		IF stReciveData.iLength > 0 THEN
			MEMSET(ADR(sReciveMessage),0,SIZEOF(sReciveMessage));
			FUN_TcpBufferDataToString(ADR(sReciveMessage),ADR(stReciveData));
			MEMCPY(ADR(sLastStatusCode),ADR(sReciveMessage),2);
			iLastStatusCode := STRING_TO_INT(sLastStatusCode);
			
			IF iLastStatusCode = 1 THEN 
				eCameraGetConnectionStatus := 1;
				
			ELSIF iLastStatusCode = 0 THEN
				eCameraGetConnectionStatus := 0;
				
			ELSIF iLastStatusCode = -1 THEN
				eCameraGetConnectionStatus := -1;
				
			ELSIF iLastStatusCode = -2 THEN
				eCameraGetConnectionStatus := -2;
				
			ELSIF iLastStatusCode = -6 THEN
				eCameraGetConnectionStatus := -6;
				
			END_IF	
			eCameraMethodState := CAMERA_METHOD_SEND_COMMAND;
			eCameraState := CAMERA_METHOD_DONE;

		END_IF
END_CASE
END_METHOD

METHOD PROTECTED MS_GetExpr
CASE eCameraMethodState OF
	CAMERA_METHOD_SEND_COMMAND:
		MEMSET(ADR(sSendMessage),0,SIZEOF(sSendMessage));
		sSendMessage := FUN_MergeStrings5('Get Expr ',sCellIndexExpr ,CONCAT(TO_STRING(iColumnExpr), TO_STRING(iRowExpr)), '$R$L', '');
		FUN_StringToTcpBufferData(ADR(sSendMessage),ADR(stSendData));
		
		IF fbTcpClient.MR_AppendToSendBuffer(stSendData) THEN
			eCameraMethodState := CAMERA_METHOD_RECEIVE_RESPONSE;
							
		END_IF

	CAMERA_METHOD_RECEIVE_RESPONSE:
		stReciveData := fbTcpClient.NextRecivedMessage;
		
		IF stReciveData.iLength > 0 THEN
			MEMSET(ADR(sReciveMessage),0,SIZEOF(sReciveMessage));
			FUN_TcpBufferDataToString(ADR(sReciveMessage),ADR(stReciveData));
			MEMCPY(ADR(sLastStatusCode),ADR(sReciveMessage),2);
			iLastStatusCode := STRING_TO_INT(sLastStatusCode);
			
			IF iLastStatusCode = 1 THEN 
				eCameraGetExprStatus := 1;
				
			ELSIF iLastStatusCode = 0 THEN
				eCameraGetExprStatus := 0;
				
			ELSIF iLastStatusCode = -1 THEN
				eCameraGetExprStatus := -1;
				
			ELSIF iLastStatusCode = -2 THEN
				eCameraGetExprStatus := -2;
				
			END_IF	
			eCameraMethodState := CAMERA_METHOD_SEND_COMMAND;
			eCameraState := CAMERA_METHOD_DONE;

		END_IF
END_CASE
END_METHOD

METHOD PROTECTED MS_GetFile
CASE eCameraMethodState OF
	CAMERA_METHOD_SEND_COMMAND:
		MEMSET(ADR(sSendMessage),0,SIZEOF(sSendMessage));
		sSendMessage := 'GF$R$L';
		FUN_StringToTcpBufferData(ADR(sSendMessage),ADR(stSendData));
		
		IF fbTcpClient.MR_AppendToSendBuffer(stSendData) THEN
			eCameraMethodState := CAMERA_METHOD_RECEIVE_RESPONSE;
							
		END_IF

	CAMERA_METHOD_RECEIVE_RESPONSE:
		stReciveData := fbTcpClient.NextRecivedMessage;
		
		IF stReciveData.iLength > 0 THEN
			MEMSET(ADR(sReciveMessage),0,SIZEOF(sReciveMessage));
			FUN_TcpBufferDataToString(ADR(sReciveMessage),ADR(stReciveData));
			MEMCPY(ADR(sLastStatusCode),ADR(sReciveMessage),2);
			iLastStatusCode := STRING_TO_INT(sLastStatusCode);
			
			IF iLastStatusCode = 1 THEN 
				eCameraGetFileStatus := 1;
				
			ELSIF iLastStatusCode = 0 THEN
				eCameraGetFileStatus := 0;
				
			ELSIF iLastStatusCode = -2 THEN
				eCameraGetFileStatus := -2;
				
			END_IF	
			eCameraMethodState := CAMERA_METHOD_SEND_COMMAND;
			eCameraState := CAMERA_METHOD_DONE;

		END_IF
END_CASE
END_METHOD

METHOD PROTECTED MS_GetFileList
CASE eCameraMethodState OF
	CAMERA_METHOD_SEND_COMMAND:
		MEMSET(ADR(sSendMessage),0,SIZEOF(sSendMessage));
		sSendMessage := 'Get Filelist$R$L';
		FUN_StringToTcpBufferData(ADR(sSendMessage),ADR(stSendData));
		
		IF fbTcpClient.MR_AppendToSendBuffer(stSendData) THEN
			eCameraMethodState := CAMERA_METHOD_RECEIVE_RESPONSE;
							
		END_IF

	CAMERA_METHOD_RECEIVE_RESPONSE:
		stReciveData := fbTcpClient.NextRecivedMessage;
		
		IF stReciveData.iLength > 0 THEN
			MEMSET(ADR(sReciveMessage),0,SIZEOF(sReciveMessage));
			FUN_TcpBufferDataToString(ADR(sReciveMessage),ADR(stReciveData));
			MEMCPY(ADR(sLastStatusCode),ADR(sReciveMessage),2);
			iLastStatusCode := STRING_TO_INT(sLastStatusCode);
			
			IF iLastStatusCode = 1 THEN 
				eCameraGetFileListStatus := 1;
				
			ELSIF iLastStatusCode = 0 THEN
				eCameraGetFileListStatus := 0;
				
			ELSIF iLastStatusCode = -1 THEN
				eCameraGetFileListStatus := -1;
				
			ELSIF iLastStatusCode = -2 THEN
				eCameraGetFileListStatus := -2;
				
			END_IF	
			eCameraMethodState := CAMERA_METHOD_SEND_COMMAND;
			eCameraState := CAMERA_METHOD_DONE;

		END_IF
END_CASE
END_METHOD

METHOD PROTECTED MS_GetJob
CASE eCameraMethodState OF
	CAMERA_METHOD_SEND_COMMAND:
		MEMSET(ADR(sSendMessage),0,SIZEOF(sSendMessage));
		sSendMessage := 'GJ$R$L';
		FUN_StringToTcpBufferData(ADR(sSendMessage),ADR(stSendData));
		
		IF fbTcpClient.MR_AppendToSendBuffer(stSendData) THEN
			eCameraMethodState := CAMERA_METHOD_RECEIVE_RESPONSE;
							
		END_IF

	CAMERA_METHOD_RECEIVE_RESPONSE:
		stReciveData := fbTcpClient.NextRecivedMessage;
		
		IF stReciveData.iLength > 0 THEN
			MEMSET(ADR(sReciveMessage),0,SIZEOF(sReciveMessage));
			FUN_TcpBufferDataToString(ADR(sReciveMessage),ADR(stReciveData));
			MEMCPY(ADR(sLastStatusCode),ADR(sReciveMessage),2);
			iLastStatusCode := STRING_TO_INT(sLastStatusCode);
			
			IF iLastStatusCode = 1 THEN 
				eCameraGetJobStatus := 1;
				
			ELSIF iLastStatusCode = 0 THEN
				eCameraGetJobStatus := 0;
				
			ELSIF iLastStatusCode = -2 THEN
				eCameraGetJobStatus := -2;
				
			END_IF	
			eCameraMethodState := CAMERA_METHOD_SEND_COMMAND;
			eCameraState := CAMERA_METHOD_DONE;

		END_IF
END_CASE
END_METHOD

METHOD PROTECTED MS_GetOnline
CASE eCameraMethodState OF
	CAMERA_METHOD_SEND_COMMAND:
		MEMSET(ADR(sSendMessage),0,SIZEOF(sSendMessage));
		sSendMessage := 'GO$R$L';
		FUN_StringToTcpBufferData(ADR(sSendMessage),ADR(stSendData));
		
		IF fbTcpClient.MR_AppendToSendBuffer(stSendData) THEN
			eCameraMethodState := CAMERA_METHOD_RECEIVE_RESPONSE;
							
		END_IF

	CAMERA_METHOD_RECEIVE_RESPONSE:
		stReciveData := fbTcpClient.NextRecivedMessage;
		
		IF stReciveData.iLength > 0 THEN
			MEMSET(ADR(sReciveMessage),0,SIZEOF(sReciveMessage));
			FUN_TcpBufferDataToString(ADR(sReciveMessage),ADR(stReciveData));
			MEMCPY(ADR(sLastStatusCode),ADR(sReciveMessage),2);
			iLastStatusCode := STRING_TO_INT(sLastStatusCode);
			
			IF iLastStatusCode = 0 THEN 
				eCameraGetOnlineStatus := 0;
				
			ELSIF iLastStatusCode = 1 THEN
				eCameraGetOnlineStatus := 1;
				
			END_IF	
			eCameraMethodState := CAMERA_METHOD_SEND_COMMAND;
			eCameraState := CAMERA_METHOD_DONE;

		END_IF
END_CASE
END_METHOD

METHOD PROTECTED MS_GetPosition
CASE eCameraGetPositionState OF
	CAMERA_GET_POSITION_SEND_COMMAND_X:
		MEMSET(ADR(sSendMessage),0,SIZEOF(sSendMessage));
		sSendMessage := FUN_MergeStrings3('GV', sPositionXVariable,'$R$L');
		FUN_StringToTcpBufferData(ADR(sSendMessage),ADR(stSendData));
		
		IF fbTcpClient.MR_AppendToSendBuffer(stSendData) THEN
			eCameraGetPositionState := CAMERA_GET_POSITION_RECEIVE_RESPONSE_X;
							
		END_IF

	CAMERA_GET_POSITION_RECEIVE_RESPONSE_X:
		stReciveData := fbTcpClient.NextRecivedMessage;
		
		IF stReciveData.iLength > 0 THEN
			MEMSET(ADR(sReciveMessage),0,SIZEOF(sReciveMessage));
			FUN_TcpBufferDataToString(ADR(sReciveMessage),ADR(stReciveData));
			MEMCPY(ADR(sLastStatusCode),ADR(sReciveMessage),2);
			iLastStatusCode := STRING_TO_INT(sLastStatusCode);
			
			IF iLastStatusCode = 1 THEN 
				eCameraGetPositionStatus := 1;
				sPositionString := TO_STRING(sReciveMessage);
				sPositionStringDel := DELETE(sPositionString,3,1);
				lrPositionX := STRING_TO_LREAL(sPositionStringDel);
				
			ELSIF iLastStatusCode = 0 THEN
				eCameraGetPositionStatus := 0;
				
			ELSIF iLastStatusCode = -1 THEN
				eCameraGetPositionStatus := -1;
				
			ELSIF iLastStatusCode = -2 THEN
				eCameraGetPositionStatus := -2;
				
			END_IF	
			eCameraGetPositionState := CAMERA_GET_POSITION_SEND_COMMAND_Y;

		END_IF
	
	CAMERA_GET_POSITION_SEND_COMMAND_Y:
		MEMSET(ADR(sSendMessage),0,SIZEOF(sSendMessage));
		sSendMessage := FUN_MergeStrings3('GV', sPositionYVariable,'$R$L');
		FUN_StringToTcpBufferData(ADR(sSendMessage),ADR(stSendData));
		
		IF fbTcpClient.MR_AppendToSendBuffer(stSendData) THEN
			eCameraGetPositionState := CAMERA_GET_POSITION_RECEIVE_RESPONSE_Y;
							
		END_IF

	CAMERA_GET_POSITION_RECEIVE_RESPONSE_Y:
		stReciveData := fbTcpClient.NextRecivedMessage;
		
		IF stReciveData.iLength > 0 THEN
			MEMSET(ADR(sReciveMessage),0,SIZEOF(sReciveMessage));
			FUN_TcpBufferDataToString(ADR(sReciveMessage),ADR(stReciveData));
			MEMCPY(ADR(sLastStatusCode),ADR(sReciveMessage),2);
			iLastStatusCode := STRING_TO_INT(sLastStatusCode);
			
			IF iLastStatusCode = 1 THEN 
				eCameraGetPositionStatus := 1;
				sPositionString := TO_STRING(sReciveMessage);
				sPositionStringDel := DELETE(sPositionString,3,1);
				lrPositionY := STRING_TO_LREAL(sPositionStringDel);
				
			ELSIF iLastStatusCode = 0 THEN
				eCameraGetPositionStatus := 0;
				
			ELSIF iLastStatusCode = -1 THEN
				eCameraGetPositionStatus := -1;
				
			ELSIF iLastStatusCode = -2 THEN
				eCameraGetPositionStatus := -2;
				
			END_IF	
			eCameraGetPositionState := CAMERA_GET_POSITION_SEND_COMMAND_ROTATION;
			
		END_IF
		
		
	CAMERA_GET_POSITION_SEND_COMMAND_ROTATION:
		MEMSET(ADR(sSendMessage),0,SIZEOF(sSendMessage));
		sSendMessage := FUN_MergeStrings3('GV', sRotationVariable,'$R$L');
		FUN_StringToTcpBufferData(ADR(sSendMessage),ADR(stSendData));
		
		IF fbTcpClient.MR_AppendToSendBuffer(stSendData) THEN
			eCameraGetPositionState := CAMERA_GET_POSITION_RECEIVE_RESPONSE_ROTATION;
							
		END_IF

	CAMERA_GET_POSITION_RECEIVE_RESPONSE_ROTATION:
		stReciveData := fbTcpClient.NextRecivedMessage;
		
		IF stReciveData.iLength > 0 THEN
			MEMSET(ADR(sReciveMessage),0,SIZEOF(sReciveMessage));
			FUN_TcpBufferDataToString(ADR(sReciveMessage),ADR(stReciveData));
			MEMCPY(ADR(sLastStatusCode),ADR(sReciveMessage),2);
			iLastStatusCode := STRING_TO_INT(sLastStatusCode);
			
			IF iLastStatusCode = 1 THEN 
				eCameraGetPositionStatus := 1;
				sPositionString := TO_STRING(sReciveMessage);
				sPositionStringDel := DELETE(sPositionString,3,1);
				lrRotation := STRING_TO_LREAL(sPositionStringDel);
				
			ELSIF iLastStatusCode = 0 THEN
				eCameraGetPositionStatus := 0;
				
			ELSIF iLastStatusCode = -1 THEN
				eCameraGetPositionStatus := -1;
				
			ELSIF iLastStatusCode = -2 THEN
				eCameraGetPositionStatus := -2;
				
			END_IF	
			eCameraGetPositionState := CAMERA_GET_POSITION_GETTING_DONE;

		END_IF
		
	CAMERA_GET_POSITION_GETTING_DONE:
		IF lrPositionX = 0.0 AND lrPositionY = 0.0 THEN
			eCameraGetPositionStatus := -3;
			
		END_IF
		eCameraGetPositionState := CAMERA_GET_POSITION_SEND_COMMAND_X;
		eCameraState := CAMERA_METHOD_DONE;
		
END_CASE
END_METHOD

METHOD PROTECTED MS_GetValueEasyBuilder
CASE eCameraMethodState OF
	CAMERA_METHOD_SEND_COMMAND:
		MEMSET(ADR(sSendMessage),0,SIZEOF(sSendMessage));
		sSendMessage := FUN_MergeStrings3('GV', sEasyBuilderValueName,'$R$L');
		FUN_StringToTcpBufferData(ADR(sSendMessage),ADR(stSendData));
		
		IF fbTcpClient.MR_AppendToSendBuffer(stSendData) THEN
			eCameraMethodState := CAMERA_METHOD_RECEIVE_RESPONSE;
							
		END_IF

	CAMERA_METHOD_RECEIVE_RESPONSE:
		stReciveData := fbTcpClient.NextRecivedMessage;
		
		IF stReciveData.iLength > 0 THEN
			MEMSET(ADR(sReciveMessage),0,SIZEOF(sReciveMessage));
			FUN_TcpBufferDataToString(ADR(sReciveMessage),ADR(stReciveData));
			MEMCPY(ADR(sLastStatusCode),ADR(sReciveMessage),2);
			iLastStatusCode := STRING_TO_INT(sLastStatusCode);
			
			IF iLastStatusCode = 1 THEN 
				eCameraGetValueEasyBuilderStatus := 1;
				
			ELSIF iLastStatusCode = 0 THEN
				eCameraGetValueEasyBuilderStatus := 0;
				
			ELSIF iLastStatusCode = -1 THEN
				eCameraGetValueEasyBuilderStatus := -1;
				
			ELSIF iLastStatusCode = -2 THEN
				eCameraGetValueEasyBuilderStatus := -2;
				
			END_IF	
			eCameraMethodState := CAMERA_METHOD_SEND_COMMAND;
			eCameraState := CAMERA_METHOD_DONE;

		END_IF
END_CASE
END_METHOD

METHOD PROTECTED MS_GetValues
CASE eCameraGetValuesState OF
	CAMERA_GET_VALUES_SEND_COMMAND_VALUE_1:
		MEMSET(ADR(sSendMessage),0,SIZEOF(sSendMessage));
		sSendMessage := FUN_MergeStrings3('GV', sVariable1,'$R$L');
		FUN_StringToTcpBufferData(ADR(sSendMessage),ADR(stSendData));
		
		IF fbTcpClient.MR_AppendToSendBuffer(stSendData) THEN
			eCameraGetValuesState := CAMERA_GET_VALUES_RECEIVE_RESPONSE_VALUE_1;
							
		END_IF

	CAMERA_GET_VALUES_RECEIVE_RESPONSE_VALUE_1:
		stReciveData := fbTcpClient.NextRecivedMessage;
		
		IF stReciveData.iLength > 0 THEN
			MEMSET(ADR(sReciveMessage),0,SIZEOF(sReciveMessage));
			FUN_TcpBufferDataToString(ADR(sReciveMessage),ADR(stReciveData));
			MEMCPY(ADR(sLastStatusCode),ADR(sReciveMessage),2);
			iLastStatusCode := STRING_TO_INT(sLastStatusCode);
			
			IF iLastStatusCode = 1 THEN 
				eCameraGetValuesStatus := 1;
				sPositionString := TO_STRING(sReciveMessage);
				sPositionStringDel := DELETE(sPositionString,3,1);
				lrValue1 := STRING_TO_LREAL(sPositionStringDel);
				
			ELSIF iLastStatusCode = 0 THEN
				eCameraGetValuesStatus := 0;
				
			ELSIF iLastStatusCode = -1 THEN
				eCameraGetValuesStatus := -1;
				
			ELSIF iLastStatusCode = -2 THEN
				eCameraGetValuesStatus := -2;
				
			END_IF	
			eCameraGetValuesState := CAMERA_GET_VALUES_SEND_COMMAND_VALUE_2;

		END_IF
	
	CAMERA_GET_VALUES_SEND_COMMAND_VALUE_2:
		MEMSET(ADR(sSendMessage),0,SIZEOF(sSendMessage));
		sSendMessage := FUN_MergeStrings3('GV', sVariable2,'$R$L');
		FUN_StringToTcpBufferData(ADR(sSendMessage),ADR(stSendData));
		
		IF fbTcpClient.MR_AppendToSendBuffer(stSendData) THEN
			eCameraGetValuesState := CAMERA_GET_VALUES_RECEIVE_RESPONSE_VALUE_2;
							
		END_IF

	CAMERA_GET_VALUES_RECEIVE_RESPONSE_VALUE_2:
		stReciveData := fbTcpClient.NextRecivedMessage;
		
		IF stReciveData.iLength > 0 THEN
			MEMSET(ADR(sReciveMessage),0,SIZEOF(sReciveMessage));
			FUN_TcpBufferDataToString(ADR(sReciveMessage),ADR(stReciveData));
			MEMCPY(ADR(sLastStatusCode),ADR(sReciveMessage),2);
			iLastStatusCode := STRING_TO_INT(sLastStatusCode);
			
			IF iLastStatusCode = 1 THEN 
				eCameraGetValuesStatus := 1;
				sPositionString := TO_STRING(sReciveMessage);
				sPositionStringDel := DELETE(sPositionString,3,1);
				lrValue2 := STRING_TO_LREAL(sPositionStringDel);
				
			ELSIF iLastStatusCode = 0 THEN
				eCameraGetValuesStatus := 0;
				
			ELSIF iLastStatusCode = -1 THEN
				eCameraGetValuesStatus := -1;
				
			ELSIF iLastStatusCode = -2 THEN
				eCameraGetValuesStatus := -2;
				
			END_IF	
			eCameraGetValuesState := CAMERA_GET_VALUES_SEND_COMMAND_VALUE_3;
			
		END_IF
		
		
	CAMERA_GET_VALUES_SEND_COMMAND_VALUE_3:
		MEMSET(ADR(sSendMessage),0,SIZEOF(sSendMessage));
		sSendMessage := FUN_MergeStrings3('GV', sVariable3,'$R$L');
		FUN_StringToTcpBufferData(ADR(sSendMessage),ADR(stSendData));
		
		IF fbTcpClient.MR_AppendToSendBuffer(stSendData) THEN
			eCameraGetValuesState := CAMERA_GET_VALUES_RECEIVE_RESPONSE_VALUE_3;

		END_IF

	CAMERA_GET_VALUES_RECEIVE_RESPONSE_VALUE_3:
		stReciveData := fbTcpClient.NextRecivedMessage;
		
		IF stReciveData.iLength > 0 THEN
			MEMSET(ADR(sReciveMessage),0,SIZEOF(sReciveMessage));
			FUN_TcpBufferDataToString(ADR(sReciveMessage),ADR(stReciveData));
			MEMCPY(ADR(sLastStatusCode),ADR(sReciveMessage),2);
			iLastStatusCode := STRING_TO_INT(sLastStatusCode);
			
			IF iLastStatusCode = 1 THEN 
				eCameraGetValuesStatus := 1;
				sPositionString := TO_STRING(sReciveMessage);
				sPositionStringDel := DELETE(sPositionString,3,1);
				lrValue3 := STRING_TO_LREAL(sPositionStringDel);
				
			ELSIF iLastStatusCode = 0 THEN
				eCameraGetValuesStatus := 0;
				
			ELSIF iLastStatusCode = -1 THEN
				eCameraGetValuesStatus := -1;
				
			ELSIF iLastStatusCode = -2 THEN
				eCameraGetValuesStatus := -2;
				
			END_IF	
			eCameraGetValuesState := CAMERA_GET_VALUES_SEND_COMMAND_VALUE_4;

		END_IF


	CAMERA_GET_VALUES_SEND_COMMAND_VALUE_4:
		MEMSET(ADR(sSendMessage),0,SIZEOF(sSendMessage));
		sSendMessage := FUN_MergeStrings3('GV', sVariable4,'$R$L');
		FUN_StringToTcpBufferData(ADR(sSendMessage),ADR(stSendData));
		
		IF fbTcpClient.MR_AppendToSendBuffer(stSendData) THEN
			eCameraGetValuesState := CAMERA_GET_VALUES_RECEIVE_RESPONSE_VALUE_4;
							
		END_IF

	CAMERA_GET_VALUES_RECEIVE_RESPONSE_VALUE_4:
		stReciveData := fbTcpClient.NextRecivedMessage;
		
		IF stReciveData.iLength > 0 THEN
			MEMSET(ADR(sReciveMessage),0,SIZEOF(sReciveMessage));
			FUN_TcpBufferDataToString(ADR(sReciveMessage),ADR(stReciveData));
			MEMCPY(ADR(sLastStatusCode),ADR(sReciveMessage),2);
			iLastStatusCode := STRING_TO_INT(sLastStatusCode);
			
			IF iLastStatusCode = 1 THEN 
				eCameraGetValuesStatus := 1;
				sPositionString := TO_STRING(sReciveMessage);
				sPositionStringDel := DELETE(sPositionString,3,1);
				lrValue4 := STRING_TO_LREAL(sPositionStringDel);
				
			ELSIF iLastStatusCode = 0 THEN
				eCameraGetValuesStatus := 0;
				
			ELSIF iLastStatusCode = -1 THEN
				eCameraGetValuesStatus := -1;
				
			ELSIF iLastStatusCode = -2 THEN
				eCameraGetValuesStatus := -2;
				
			END_IF	
			eCameraGetValuesState := CAMERA_GET_VALUES_GETTING_DONE;

		END_IF
		
	CAMERA_GET_VALUES_GETTING_DONE:
		
		IF lrValue1 = 0.0 OR lrValue2 = 0.0 OR lrValue3 = 0.0 OR lrValue4 = 0.0 THEN
			eCameraGetValuesStatus := -3;
			
		END_IF
		eCameraGetValuesState := CAMERA_GET_VALUES_SEND_COMMAND_VALUE_1;
		eCameraState := CAMERA_METHOD_DONE;
		
END_CASE
END_METHOD

METHOD PROTECTED MS_GetValueSpreadsheet
CASE eCameraMethodState OF
	CAMERA_METHOD_SEND_COMMAND:
		MEMSET(ADR(sSendMessage),0,SIZEOF(sSendMessage));
		sSendMessage := FUN_MergeStrings5('GV', TO_STRING(iColumnValueSpreadsheet), TO_STRING(iRowValueSpreadsheet), '$R$L', '');
		FUN_StringToTcpBufferData(ADR(sSendMessage),ADR(stSendData));
		
		IF fbTcpClient.MR_AppendToSendBuffer(stSendData) THEN
			eCameraMethodState := CAMERA_METHOD_RECEIVE_RESPONSE;
							
		END_IF

	CAMERA_METHOD_RECEIVE_RESPONSE:
		stReciveData := fbTcpClient.NextRecivedMessage;
		
		IF stReciveData.iLength > 0 THEN
			MEMSET(ADR(sReciveMessage),0,SIZEOF(sReciveMessage));
			FUN_TcpBufferDataToString(ADR(sReciveMessage),ADR(stReciveData));
			MEMCPY(ADR(sLastStatusCode),ADR(sReciveMessage),2);
			iLastStatusCode := STRING_TO_INT(sLastStatusCode);
			
			IF iLastStatusCode = 1 THEN 
				eCameraGetValueSpreadsheetStatus := 1;
				
			ELSIF iLastStatusCode = 0 THEN
				eCameraGetValueSpreadsheetStatus := 0;
				
			ELSIF iLastStatusCode = -1 THEN
				eCameraGetValueSpreadsheetStatus := -1;
				
			ELSIF iLastStatusCode = -2 THEN
				eCameraGetValueSpreadsheetStatus := -2;
				
			END_IF	
			eCameraMethodState := CAMERA_METHOD_SEND_COMMAND;
			eCameraState := CAMERA_METHOD_DONE;

		END_IF
END_CASE
END_METHOD

METHOD PROTECTED MS_Idle
;
END_METHOD

METHOD PROTECTED MS_ImageTrigger
CASE eCameraMethodState OF
	CAMERA_METHOD_SEND_COMMAND:
		MEMSET(ADR(sSendMessage),0,SIZEOF(sSendMessage));
		sSendMessage := 'SW8$R$L';
		FUN_StringToTcpBufferData(ADR(sSendMessage),ADR(stSendData));
		
		IF fbTcpClient.MR_AppendToSendBuffer(stSendData) THEN
			eCameraMethodState := CAMERA_METHOD_RECEIVE_RESPONSE;
							
		END_IF

	CAMERA_METHOD_RECEIVE_RESPONSE:
		stReciveData := fbTcpClient.NextRecivedMessage;
		
		IF stReciveData.iLength > 0 THEN
			MEMSET(ADR(sReciveMessage),0,SIZEOF(sReciveMessage));
			FUN_TcpBufferDataToString(ADR(sReciveMessage),ADR(stReciveData));
			MEMCPY(ADR(sLastStatusCode),ADR(sReciveMessage),2);
			iLastStatusCode := STRING_TO_INT(sLastStatusCode);
			
			IF iLastStatusCode = 1 THEN 
				eCameraImageTriggerStatus := 1;
				
			ELSIF iLastStatusCode = 0 THEN
				eCameraImageTriggerStatus := 0;
				
			ELSIF iLastStatusCode = -1 THEN
				eCameraImageTriggerStatus := -1;
				
			ELSIF iLastStatusCode = -2 THEN
				eCameraImageTriggerStatus := -2;
				
			ELSIF iLastStatusCode = -6 THEN
				eCameraImageTriggerStatus := -6;
				
			END_IF	
			eCameraMethodState := CAMERA_METHOD_SEND_COMMAND;			
			eCameraState := CAMERA_METHOD_DONE;

		END_IF
END_CASE
END_METHOD

METHOD PROTECTED MS_Initializing //C:\TwinCAT\log\filelog.txt
VAR_INST
//	tClearBuffers		:	TON;
END_VAR
CASE eCameraInitState OF
	CAMERA_INIT_CONNECTION:
		fbTcpClient.MR_Init();
		
		IF fbTcpClient.Active THEN
			eCameraInitState := CAMERA_INIT_CLEAR_BUFFER;	
			
		ELSIF fbTcpClient.Error THEN
			bError := TRUE;
			iErrorID := fbTcpClient.ErrorID;
			
		END_IF
		
	CAMERA_INIT_CLEAR_BUFFER:
		fbTcpClient.MR_ClearAllBuffers();
		eCameraInitState := CAMERA_INIT_WAIT_FOR_USERNAME;
		
		IF fbTcpClient.Error THEN
			bError := TRUE;
			iErrorID := fbTcpClient.ErrorID;
			
		END_IF
		
	CAMERA_INIT_WAIT_FOR_USERNAME: 
		stReciveData := fbTcpClient.NextRecivedMessage;
		
		IF stReciveData.iLength > 0 THEN
			MEMSET(ADR(sReciveMessage),0,SIZEOF(sReciveMessage));
			FUN_TcpBufferDataToString(ADR(sReciveMessage),ADR(stReciveData));		
	
			IF RIGHT(sReciveMessage, 6) = 'User: ' THEN	
				eCameraInitState := CAMERA_INIT_WRITE_USER;
			
			END_IF
		ELSIF fbTcpClient.Error THEN
			bError := TRUE;
			iErrorID := fbTcpClient.ErrorID;
			
		END_IF
			
	CAMERA_INIT_WRITE_USER:
		MEMSET(ADR(sSendMessage),0,SIZEOF(sSendMessage));
		sSendMessage := 'admin$R$L';
		FUN_StringToTcpBufferData(ADR(sSendMessage),ADR(stSendData));
		stSendData.iLength := INT_TO_UDINT(LEN(sSendMessage));
		
		IF fbTcpClient.MR_AppendToSendBuffer(stSendData) THEN
			eCameraInitState := CAMERA_INIT_WAIT_FOR_PASSWORD;
		
		ELSIF fbTcpClient.Error THEN
			bError := TRUE;
			iErrorID := fbTcpClient.ErrorID;
			
		END_IF
		
	CAMERA_INIT_WAIT_FOR_PASSWORD:
		stReciveData := fbTcpClient.NextRecivedMessage;
		
		IF stReciveData.iLength > 0 THEN
			MEMSET(ADR(sReciveMessage),0,SIZEOF(sReciveMessage));
			FUN_TcpBufferDataToString(ADR(sReciveMessage),ADR(stReciveData));
			
			IF sReciveMessage = 'Password: ' THEN		
				eCameraInitState := CAMERA_INIT_WRITE_PASSWORD;
			
			END_IF
		ELSIF fbTcpClient.Error THEN
			bError := TRUE;
			iErrorID := fbTcpClient.ErrorID;
			
		END_IF

	CAMERA_INIT_WRITE_PASSWORD:
		MEMSET(ADR(sSendMessage),0,SIZEOF(sSendMessage));
		sSendMessage := '$R$L';
		FUN_StringToTcpBufferData(ADR(sSendMessage),ADR(stSendData));
		stSendData.iLength := INT_TO_UDINT(LEN(sSendMessage));
		
		IF fbTcpClient.MR_AppendToSendBuffer(stSendData) THEN
			eCameraInitState := CAMERA_INIT_WAIT_FOR_CONFIRMATION;

		ELSIF fbTcpClient.Error THEN
			bError := TRUE;
			iErrorID := fbTcpClient.ErrorID;
			
		END_IF
		
	CAMERA_INIT_WAIT_FOR_CONFIRMATION:
		stReciveData := fbTcpClient.NextRecivedMessage;
		
		IF stReciveData.iLength > 0 THEN
			MEMSET(ADR(sReciveMessage),0,SIZEOF(sReciveMessage));
			FUN_TcpBufferDataToString(ADR(sReciveMessage),ADR(stReciveData));
	
			IF sReciveMessage = 'User Logged In$R$L' THEN		
				eCameraInitState := CAMERA_INIT_DONE;
			
			END_IF
		ELSIF fbTcpClient.Error THEN
			bError := TRUE;
			iErrorID := fbTcpClient.ErrorID;
			
		END_IF
		
	CAMERA_INIT_DONE:
		eCameraInitState := CAMERA_INIT_CONNECTION;
		eCameraState := CAMERA_READY;
			
END_CASE
END_METHOD

METHOD PROTECTED MS_LoadFile
CASE eCameraMethodState OF
	CAMERA_METHOD_SEND_COMMAND:
		MEMSET(ADR(sSendMessage),0,SIZEOF(sSendMessage));
		sSendMessage := FUN_MergeStrings3('LF', sLoadFileName,'$R$L');
		FUN_StringToTcpBufferData(ADR(sSendMessage),ADR(stSendData));
		
		IF fbTcpClient.MR_AppendToSendBuffer(stSendData) THEN
			eCameraMethodState := CAMERA_METHOD_RECEIVE_RESPONSE;
							
		END_IF

	CAMERA_METHOD_RECEIVE_RESPONSE:
		stReciveData := fbTcpClient.NextRecivedMessage;
		
		IF stReciveData.iLength > 0 THEN
			MEMSET(ADR(sReciveMessage),0,SIZEOF(sReciveMessage));
			FUN_TcpBufferDataToString(ADR(sReciveMessage),ADR(stReciveData));
			MEMCPY(ADR(sLastStatusCode),ADR(sReciveMessage),2);
			iLastStatusCode := STRING_TO_INT(sLastStatusCode);
			
			IF iLastStatusCode = 1 THEN 
				eCameraLoadFileStatus := 1;
				
			ELSIF iLastStatusCode = 0 THEN
				eCameraLoadFileStatus := 0;
				
			ELSIF iLastStatusCode = -1 THEN
				eCameraLoadFileStatus := -1;
				
			ELSIF iLastStatusCode = -2 THEN
				eCameraLoadFileStatus := -2;
				
			ELSIF iLastStatusCode = -4 THEN
				eCameraLoadFileStatus := -4;
				
			ELSIF iLastStatusCode = -6 THEN
				eCameraLoadFileStatus := -6;
				
			END_IF	
			eCameraMethodState := CAMERA_METHOD_SEND_COMMAND;
			eCameraState := CAMERA_METHOD_DONE;

		END_IF
END_CASE
END_METHOD

METHOD PROTECTED MS_MethodDone
VAR_INPUT
END_VAR
IF NOT bBusy THEN
	eCameraState := CAMERA_IDLE;
	
END_IF
END_METHOD

METHOD PROTECTED MS_PutLive
CASE eCameraMethodState OF
	CAMERA_METHOD_SEND_COMMAND:
		MEMSET(ADR(sSendMessage),0,SIZEOF(sSendMessage));
		sSendMessage := FUN_MergeStrings3('Put live ', TO_STRING(bEnableLiveAcquisition), '$R$L');
		FUN_StringToTcpBufferData(ADR(sSendMessage),ADR(stSendData));
		
		IF fbTcpClient.MR_AppendToSendBuffer(stSendData) THEN
			eCameraMethodState := CAMERA_METHOD_RECEIVE_RESPONSE;
							
		END_IF

	CAMERA_METHOD_RECEIVE_RESPONSE:
		stReciveData := fbTcpClient.NextRecivedMessage;
		
		IF stReciveData.iLength > 0 THEN
			MEMSET(ADR(sReciveMessage),0,SIZEOF(sReciveMessage));
			FUN_TcpBufferDataToString(ADR(sReciveMessage),ADR(stReciveData));
			MEMCPY(ADR(sLastStatusCode),ADR(sReciveMessage),2);
			iLastStatusCode := STRING_TO_INT(sLastStatusCode);
			
			IF iLastStatusCode = 1 THEN 
				eCameraPutLiveStatus := 1;
				
			ELSIF iLastStatusCode = 0 THEN
				eCameraPutLiveStatus := 0;
				
			ELSIF iLastStatusCode = -1 THEN
				eCameraPutLiveStatus := -1;
				
			ELSIF iLastStatusCode = -2 THEN
				eCameraPutLiveStatus := -2;
				
			ELSIF iLastStatusCode = -6 THEN
				eCameraPutLiveStatus := -6;
				
			END_IF	
			eCameraMethodState := CAMERA_METHOD_SEND_COMMAND;
			eCameraState := CAMERA_METHOD_DONE;

		END_IF
END_CASE
END_METHOD

METHOD PROTECTED MS_PutPortnum
CASE eCameraMethodState OF
	CAMERA_METHOD_SEND_COMMAND:
		MEMSET(ADR(sSendMessage),0,SIZEOF(sSendMessage));
		sSendMessage := FUN_MergeStrings3('Put Portnum ', TO_STRING(iPortNumber), '$R$L');
		FUN_StringToTcpBufferData(ADR(sSendMessage),ADR(stSendData));
		
		IF fbTcpClient.MR_AppendToSendBuffer(stSendData) THEN
			eCameraMethodState := CAMERA_METHOD_RECEIVE_RESPONSE;
							
		END_IF

	CAMERA_METHOD_RECEIVE_RESPONSE:
		stReciveData := fbTcpClient.NextRecivedMessage;
		
		IF stReciveData.iLength > 0 THEN
			MEMSET(ADR(sReciveMessage),0,SIZEOF(sReciveMessage));
			FUN_TcpBufferDataToString(ADR(sReciveMessage),ADR(stReciveData));
			MEMCPY(ADR(sLastStatusCode),ADR(sReciveMessage),2);
			iLastStatusCode := STRING_TO_INT(sLastStatusCode);
			
			IF iLastStatusCode = 1 THEN 
				eCameraPutPortnumStatus := 1;
				
			ELSIF iLastStatusCode = 0 THEN
				eCameraPutPortnumStatus := 0;
				
			ELSIF iLastStatusCode = -1 THEN
				eCameraPutPortnumStatus := -1;
				
			ELSIF iLastStatusCode = -2 THEN
				eCameraPutPortnumStatus := -2;
				
			ELSIF iLastStatusCode = -6 THEN
				eCameraPutPortnumStatus := -6;
				
			END_IF	
			eCameraMethodState := CAMERA_METHOD_SEND_COMMAND;
			eCameraState := CAMERA_METHOD_DONE;

		END_IF
END_CASE
END_METHOD

METHOD PROTECTED MS_PutTimeout
CASE eCameraMethodState OF
	CAMERA_METHOD_SEND_COMMAND:
		MEMSET(ADR(sSendMessage),0,SIZEOF(sSendMessage));
		sSendMessage := FUN_MergeStrings3('Put Timeout ', TO_STRING(iTimeout), '$R$L');
		FUN_StringToTcpBufferData(ADR(sSendMessage),ADR(stSendData));
		
		IF fbTcpClient.MR_AppendToSendBuffer(stSendData) THEN
			eCameraMethodState := CAMERA_METHOD_RECEIVE_RESPONSE;
							
		END_IF

	CAMERA_METHOD_RECEIVE_RESPONSE:
		stReciveData := fbTcpClient.NextRecivedMessage;
		
		IF stReciveData.iLength > 0 THEN
			MEMSET(ADR(sReciveMessage),0,SIZEOF(sReciveMessage));
			FUN_TcpBufferDataToString(ADR(sReciveMessage),ADR(stReciveData));
			MEMCPY(ADR(sLastStatusCode),ADR(sReciveMessage),2);
			iLastStatusCode := STRING_TO_INT(sLastStatusCode);
			
			IF iLastStatusCode = 1 THEN 
				eCameraPutTimeoutStatus := 1;
				
			ELSIF iLastStatusCode = 0 THEN
				eCameraPutTimeoutStatus := 0;
				
			ELSIF iLastStatusCode = -1 THEN
				eCameraPutTimeoutStatus := -1;
				
			ELSIF iLastStatusCode = -6 THEN
				eCameraPutTimeoutStatus := -6;
				
			END_IF	
			eCameraMethodState := CAMERA_METHOD_SEND_COMMAND;
			eCameraState := CAMERA_METHOD_DONE;
			
		END_IF
END_CASE
END_METHOD

METHOD PROTECTED MS_PutUpdate
CASE eCameraMethodState OF
	CAMERA_METHOD_SEND_COMMAND:
		MEMSET(ADR(sSendMessage),0,SIZEOF(sSendMessage));
		sSendMessage := FUN_MergeStrings3('Put Update ', TO_STRING(iUpdateNumber), '$R$L');
		FUN_StringToTcpBufferData(ADR(sSendMessage),ADR(stSendData));
		
		IF fbTcpClient.MR_AppendToSendBuffer(stSendData) THEN
			eCameraMethodState := CAMERA_METHOD_RECEIVE_RESPONSE;
							
		END_IF

	CAMERA_METHOD_RECEIVE_RESPONSE:
		stReciveData := fbTcpClient.NextRecivedMessage;
		
		IF stReciveData.iLength > 0 THEN
			MEMSET(ADR(sReciveMessage),0,SIZEOF(sReciveMessage));
			FUN_TcpBufferDataToString(ADR(sReciveMessage),ADR(stReciveData));
			MEMCPY(ADR(sLastStatusCode),ADR(sReciveMessage),2);
			iLastStatusCode := STRING_TO_INT(sLastStatusCode);
			
			IF iLastStatusCode = 1 THEN 
				eCameraPutUpdateStatus := 1;
				
			ELSIF iLastStatusCode = 0 THEN
				eCameraPutUpdateStatus := 0;
				
			ELSIF iLastStatusCode = -1 THEN
				eCameraPutUpdateStatus := -1;
				
			ELSIF iLastStatusCode = -2 THEN
				eCameraPutUpdateStatus := -2;
				
			ELSIF iLastStatusCode = -6 THEN
				eCameraPutUpdateStatus := -6;
				
			END_IF	
			eCameraMethodState := CAMERA_METHOD_SEND_COMMAND;
			eCameraState := CAMERA_METHOD_DONE;

		END_IF
END_CASE
END_METHOD

METHOD PROTECTED MS_PutWatch
CASE eCameraMethodState OF
	CAMERA_METHOD_SEND_COMMAND:
		MEMSET(ADR(sSendMessage),0,SIZEOF(sSendMessage));
		sSendMessage := FUN_MergeStrings5('Put Watch ', TO_STRING(iColumnPut), TO_STRING(iRowPut), TO_STRING(iOutputEnable), '$R$L');
		FUN_StringToTcpBufferData(ADR(sSendMessage),ADR(stSendData));
		
		IF fbTcpClient.MR_AppendToSendBuffer(stSendData) THEN
			eCameraMethodState := CAMERA_METHOD_RECEIVE_RESPONSE;
							
		END_IF

	CAMERA_METHOD_RECEIVE_RESPONSE:
		stReciveData := fbTcpClient.NextRecivedMessage;
		
		IF stReciveData.iLength > 0 THEN
			MEMSET(ADR(sReciveMessage),0,SIZEOF(sReciveMessage));
			FUN_TcpBufferDataToString(ADR(sReciveMessage),ADR(stReciveData));
			MEMCPY(ADR(sLastStatusCode),ADR(sReciveMessage),2);
			iLastStatusCode := STRING_TO_INT(sLastStatusCode);
			
			IF iLastStatusCode = 1 THEN 
				eCameraPutWatchStatus := 1;
				
			ELSIF iLastStatusCode = 0 THEN
				eCameraPutWatchStatus := 0;
				
			ELSIF iLastStatusCode = -1 THEN
				eCameraPutWatchStatus := -1;
				
			ELSIF iLastStatusCode = -2 THEN
				eCameraPutWatchStatus := -2;
				
			ELSIF iLastStatusCode = -6 THEN
				eCameraPutWatchStatus := -6;
				
			END_IF	
			eCameraMethodState := CAMERA_METHOD_SEND_COMMAND;
			eCameraState := CAMERA_METHOD_DONE;

		END_IF
END_CASE
END_METHOD

METHOD PROTECTED MS_Ready
VAR_INPUT
END_VAR
eCameraState := CAMERA_IDLE;
END_METHOD

METHOD PROTECTED MS_Reset
VAR_INPUT
END_VAR
IF M_ResetParameters() THEN
	eCameraState := CAMERA_METHOD_DONE;
	
END_IF
END_METHOD

METHOD PROTECTED MS_ResetSystem
CASE eCameraMethodState OF
	CAMERA_METHOD_SEND_COMMAND:
		MEMSET(ADR(sSendMessage),0,SIZEOF(sSendMessage));
		sSendMessage := 'RT$R$L';
		FUN_StringToTcpBufferData(ADR(sSendMessage),ADR(stSendData));
		
		IF fbTcpClient.MR_AppendToSendBuffer(stSendData) THEN
			eCameraMethodState := CAMERA_METHOD_RECEIVE_RESPONSE;
							
		END_IF

	CAMERA_METHOD_RECEIVE_RESPONSE:
		stReciveData := fbTcpClient.NextRecivedMessage;
		
		IF stReciveData.iLength > 0 THEN
			MEMSET(ADR(sReciveMessage),0,SIZEOF(sReciveMessage));
			FUN_TcpBufferDataToString(ADR(sReciveMessage),ADR(stReciveData));
			MEMCPY(ADR(sLastStatusCode),ADR(sReciveMessage),2);
			iLastStatusCode := STRING_TO_INT(sLastStatusCode);
			
			IF iLastStatusCode = -6 THEN 
				eCameraResetSystemStatus := -6;
				
			END_IF	
		ELSE
			eCameraResetSystemStatus := -1;
			
		END_IF
		eCameraMethodState := CAMERA_METHOD_SEND_COMMAND;
		eCameraState := CAMERA_METHOD_DONE;
		
END_CASE
END_METHOD

METHOD PROTECTED MS_SetJob
CASE eCameraMethodState OF
	CAMERA_METHOD_SEND_COMMAND:
		MEMSET(ADR(sSendMessage),0,SIZEOF(sSendMessage));
		sSendMessage := FUN_MergeStrings3('SJ', TO_STRING(iJobNumber), '$R$L');
		FUN_StringToTcpBufferData(ADR(sSendMessage),ADR(stSendData));
		
		IF fbTcpClient.MR_AppendToSendBuffer(stSendData) THEN
			eCameraMethodState := CAMERA_METHOD_RECEIVE_RESPONSE;
							
		END_IF

	CAMERA_METHOD_RECEIVE_RESPONSE:
		stReciveData := fbTcpClient.NextRecivedMessage;
		
		IF stReciveData.iLength > 0 THEN
			MEMSET(ADR(sReciveMessage),0,SIZEOF(sReciveMessage));
			FUN_TcpBufferDataToString(ADR(sReciveMessage),ADR(stReciveData));
			MEMCPY(ADR(sLastStatusCode),ADR(sReciveMessage),2);
			iLastStatusCode := STRING_TO_INT(sLastStatusCode);
			
			IF iLastStatusCode = 1 THEN 
				eCameraSetJobStatus := 1;
				
			ELSIF iLastStatusCode = 0 THEN
				eCameraSetJobStatus := 0;
				
			ELSIF iLastStatusCode = -1 THEN
				eCameraSetJobStatus := -1;
				
			ELSIF iLastStatusCode = -2 THEN
				eCameraSetJobStatus := -2;
				
			ELSIF iLastStatusCode = -4 THEN
				eCameraSetJobStatus := -4;
				
			ELSIF iLastStatusCode = -6 THEN
				eCameraSetJobStatus := -6;
				
			END_IF	
			eCameraMethodState := CAMERA_METHOD_SEND_COMMAND;
			eCameraState := CAMERA_METHOD_DONE;

		END_IF
END_CASE
END_METHOD

METHOD PROTECTED MS_SetOnline
CASE eCameraMethodState OF
	CAMERA_METHOD_SEND_COMMAND:
		MEMSET(ADR(sSendMessage),0,SIZEOF(sSendMessage));
		sSendMessage := FUN_MergeStrings3('SO', TO_STRING(bSetCameraOnline), '$R$L');
		FUN_StringToTcpBufferData(ADR(sSendMessage),ADR(stSendData));
		
		IF fbTcpClient.MR_AppendToSendBuffer(stSendData) THEN
			eCameraMethodState := CAMERA_METHOD_RECEIVE_RESPONSE;
							
		END_IF

	CAMERA_METHOD_RECEIVE_RESPONSE:
		stReciveData := fbTcpClient.NextRecivedMessage;
		
		IF stReciveData.iLength > 0 THEN
			MEMSET(ADR(sReciveMessage),0,SIZEOF(sReciveMessage));
			FUN_TcpBufferDataToString(ADR(sReciveMessage),ADR(stReciveData));
			MEMCPY(ADR(sLastStatusCode),ADR(sReciveMessage),2);
			iLastStatusCode := STRING_TO_INT(sLastStatusCode);
			
			IF iLastStatusCode = 1 THEN 
				eCameraSetOnlineStatus := 1;
				
			ELSIF iLastStatusCode = 0 THEN
				eCameraSetOnlineStatus := 0;
				
			ELSIF iLastStatusCode = -1 THEN
				eCameraSetOnlineStatus := -1;
				
			ELSIF iLastStatusCode = -2 THEN
				eCameraSetOnlineStatus := -2;
				
			ELSIF iLastStatusCode = -5 THEN
				eCameraSetOnlineStatus := -5;
				
			ELSIF iLastStatusCode = -6 THEN
				eCameraSetOnlineStatus := -6;
				
			END_IF	
			eCameraMethodState := CAMERA_METHOD_SEND_COMMAND;
			eCameraState := CAMERA_METHOD_DONE;

		END_IF
END_CASE
END_METHOD

METHOD PROTECTED MS_StoreFile
CASE eCameraMethodState OF
	CAMERA_METHOD_SEND_COMMAND:
		MEMSET(ADR(sSendMessage),0,SIZEOF(sSendMessage));
		sSendMessage := FUN_MergeStrings3('TF', sStoreFileName,'$R$L');
		FUN_StringToTcpBufferData(ADR(sSendMessage),ADR(stSendData));
		
		IF fbTcpClient.MR_AppendToSendBuffer(stSendData) THEN
			eCameraMethodState := CAMERA_METHOD_RECEIVE_RESPONSE;
							
		END_IF

	CAMERA_METHOD_RECEIVE_RESPONSE:
		stReciveData := fbTcpClient.NextRecivedMessage;
		
		IF stReciveData.iLength > 0 THEN
			MEMSET(ADR(sReciveMessage),0,SIZEOF(sReciveMessage));
			FUN_TcpBufferDataToString(ADR(sReciveMessage),ADR(stReciveData));
			MEMCPY(ADR(sLastStatusCode),ADR(sReciveMessage),2);
			iLastStatusCode := STRING_TO_INT(sLastStatusCode);
			
			IF iLastStatusCode = 1 THEN 
				eCameraStoreFileStatus := 1;
			ELSIF iLastStatusCode = 0 THEN
				eCameraStoreFileStatus := 0;
			ELSIF iLastStatusCode = -1 THEN
				eCameraStoreFileStatus := -1;
			ELSIF iLastStatusCode = -2 THEN
				eCameraStoreFileStatus := -2;
			ELSIF iLastStatusCode = -6 THEN
				eCameraStoreFileStatus := -6;
			END_IF	
			eCameraMethodState := CAMERA_METHOD_SEND_COMMAND;
			eCameraState := CAMERA_METHOD_DONE;

		END_IF
END_CASE
END_METHOD

METHOD PROTECTED MS_Uninitialized
;
END_METHOD

PROPERTY Name : STRING
GET
Name := sName;
END_GET
SET
sName := Name;
END_SET
END_PROPERTY

PROPERTY ref_TcpClient : REFERENCE TO FB_TcpClient
GET
ref_TcpClient REF= fbTcpClient;
END_GET
END_PROPERTY

METHOD PROTECTED StateMachine
CASE eCameraState OF
	CAMERA_UNINITIALIZED:
		MS_Uninitialized();
		
	CAMERA_INITIALIZING:
		MS_Initializing();
		
	CAMERA_READY:
		MS_Ready();
	
	CAMERA_IDLE:
		MS_Idle();	
		
	CAMERA_RESET:
		MS_Reset();
		
	CAMERA_LOAD_FILE:
		MS_LoadFile();	
		
	CAMERA_GET_FILE:
		MS_GetFile();

	CAMERA_GET_VALUE_EASY_BUILDER:
		MS_GetValueEasyBuilder();	
		
	CAMERA_GET_VALUE_SPREADSHEET:
		MS_GetValueSpreadsheet();	
		
	CAMERA_SET_ONLINE:
		MS_SetOnline();	
	
	CAMERA_GET_ONLINE:
		MS_GetOnline();
		
	CAMERA_RESET_SYSTEM:
		MS_ResetSystem();
	
	CAMERA_GET_CONNECTIONS:
		MS_GetConnections();
		
	CAMERA_GET_EXPR:
		MS_GetExpr();
	
	CAMERA_GET_FILE_LIST:
		MS_GetFileList();
	
	CAMERA_PUT_LIVE:
		MS_PutLive();
	
	CAMERA_PUT_PORTNUM:
		MS_PutPortnum();
	
	CAMERA_PUT_TIMEOUT:
		MS_PutTimeout();
	
	CAMERA_PUT_UPDATE:
		MS_PutUpdate();
	
	CAMERA_PUT_WATCH:
		MS_PutWatch();	
	
	CAMERA_SET_JOB:
		MS_SetJob();
		
	CAMERA_GET_JOB:
		MS_GetJob();
	
	CAMERA_STORE_FILE:
		MS_StoreFile();	
		
	CAMERA_GET_POSITION:
		MS_GetPosition();
	
	CAMERA_IMAGE_TRIGGER:
		MS_ImageTrigger();
	
	CAMERA_GET_VALUES:
		MS_GetValues();
	
	CAMERA_METHOD_DONE:
		MS_MethodDone();
	
	CAMERA_ABORTING:
		MS_Aborting();
	
END_CASE
END_METHOD

END_FUNCTION_BLOCK

// ---- POUs/Machine/Visu Control/F_CloseDialog_1.TcPOU
FUNCTION F_CloseDialog_1 : BOOL
VAR_INPUT
	sDialogName : STRING;
END_VAR
VAR
	pstClientData : POINTER TO VisuElems.VisuStructClientData;
	itfDialogManager : VisuElems.IDialogManager;
	itfMyDialog : VisuElems.IVisualisationDialog;
	stVisuRect : VisuElems.VisuStructSimpleRectangle;
END_VAR

VisuElems.VisuElemBase.g_ClientManager.BeginIteration();
pstClientData := VisuElems.VisuElemBase.g_ClientManager.GetNextClient();
WHILE pstClientData <> 0 DO
   IF pstClientData^.GlobalData.ClientType = VisuElems.Visu_ClientType.HMITargetVisualization THEN
      itfDialogManager := VisuElems.g_VisuManager.GetDialogManager();
      itfMyDialog := itfDialogManager.GetDialog(sDialogName);
      itfDialogManager.CloseDialog	(itfMyDialog, pstClientData);
   END_IF
   pstClientData := VisuElems.VisuElemBase.g_ClientManager.GetNextClient();
END_WHILE

END_FUNCTION

// ---- POUs/Machine/Visu Control/F_OpenDialog_1.TcPOU
FUNCTION F_OpenDialog_1 : BOOL
VAR_INPUT
	sDialogName : STRING;
END_VAR
VAR
	pstClientData : POINTER TO VisuElems.VisuStructClientData;
	itfDialogManager : VisuElems.IDialogManager;
	itfMyDialog : VisuElems.IVisualisationDialog;
	stVisuRect : VisuElems.VisuStructSimpleRectangle;
END_VAR

VisuElems.VisuElemBase.g_ClientManager.BeginIteration();
pstClientData := VisuElems.VisuElemBase.g_ClientManager.GetNextClient();
WHILE pstClientData <> 0 DO
   IF pstClientData^.GlobalData.ClientType = VisuElems.Visu_ClientType.HMITargetVisualization THEN
      itfDialogManager := VisuElems.g_VisuManager.GetDialogManager();
      itfMyDialog := itfDialogManager.GetDialog(sDialogName);
      stVisuRect.ptTopLeft.iX := ANY_TO_INT(INT#0);
      stVisuRect.ptTopLeft.iY := ANY_TO_INT(INT#0);
      stVisuRect.ptBottomRight.iX := ANY_TO_INT(10);
      stVisuRect.ptBottomRight.iY := ANY_TO_INT(10);
      itfDialogManager.OpenDialog(itfMyDialog, pstClientData, FALSE, ADR(stVisuRect));
   END_IF
   pstClientData := VisuElems.VisuElemBase.g_ClientManager.GetNextClient();
END_WHILE

END_FUNCTION

// ---- GlobalTextList.TcGTLO
TEXTLIST GlobalTextList
  224 = '%2d'
  1044 = '%3.0f'
  21 = '%6.3f'
  331 = '%d'
  890 = '%f'
  976 = '%s'
  2051 = '/'
  887 = 'Abort'
  494 = 'Acceleration:'
  3798 = 'Action number:'
  487 = 'Active Alarms'
  1711 = 'Active alarms:'
  649 = 'Active critical'
  1670 = 'Active critical alarms:'
  202 = 'Active criticals:'
  709 = 'Active errors'
  780 = 'Active errors:'
  700 = 'Active warnings:'
  582 = 'Active warrnings'
  706 = 'Active warrnings:'
  370 = 'Actual Position:'
  78 = 'Actual Velocity'
  1000 = 'Admin'
  431 = 'Alarms'
  813 = 'All active alarms:'
  427 = 'Auto mode'
  931 = 'Axes'
  913 = 'Axis'
  542 = 'Back'
  300 = 'Backup'
  2292 = 'Backup and restore from external directory'
  2272 = 'Battery low'
  662 = 'Battery reset'
  917 = 'Change pass.'
  1549 = 'Clear all'
  349 = 'Clear All Alarms'
  277 = 'Close'
  410 = 'Close HMI'
  1072 = 'Commands'
  1156 = 'Controller'
  2906 = 'Controller reset'
  1047 = 'Create'
  2909 = 'Create new recipe:'
  2120 = 'Current value'
  2043 = 'Cycle pause'
  3558 = 'Cycle restore'
  2070 = 'Cycle stop'
  424 = 'Cylinders'
  1092 = 'Deceleration:'
  362 = 'Deinitialization in progress...'
  1655 = 'Digital Inputs'
  1456 = 'Digital inputs'
  1692 = 'Digital Outputs'
  1445 = 'Digital outputs'
  1090 = 'Digital outputs and valves'
  538 = 'Door Lock'
  1643 = 'Enable simulation'
  1468 = 'Error'
  2782 = 'Error reset'
  537 = 'Error: %d'
  1738 = 'Error: %s'
  368 = 'Event history'
  1107 = 'Event history:'
  86 = 'Event ID'
  619 = 'Event Text'
  297 = 'Event Type'
  77 = 'Export to file'
  1073 = 'Finishing initialization...'
  1696 = 'Force Input Value'
  244 = 'Go %s'
  2687 = 'Go auto'
  66 = 'Go home'
  1163 = 'Halt'
  2141 = 'Halted'
  110 = 'Home'
  1505 = 'Homed'
  2548 = 'In Position'
  371 = 'Initialize'
  1488 = 'Initialized'
  312 = 'Inputs'
  2436 = 'Jog'
  18 = 'Jog +'
  19 = 'Jog -'
  2152 = 'Jog mode:'
  121 = 'Lag error:'
  715 = 'Lights'
  1263 = 'Load from file'
  1426 = 'Loaded recipe'
  332 = 'Log In'
  198 = 'Log Out'
  1506 = 'Logged user'
  921 = 'Machine nearly ready to work...'
  665 = 'Machine state'
  428 = 'Manual'
  485 = 'Manual Axis Control'
  1020 = 'Manual Cylinders Control'
  822 = 'Manual mode'
  3024 = 'Manual Robots Control'
  729 = 'Mode switch'
  417 = 'Motors'
  1606 = 'Next'
  1023 = 'None'
  1645 = 'Number of:'
  1015 = 'Operator'
  1972 = 'Others'
  613 = 'Outputs'
  639 = 'Override:'
  1319 = 'Override: %2.0d'
  407 = 'Override: %2d'
  1429 = 'Override: %3.0f'
  1146 = 'Parameters:'
  1309 = 'Path:'
  725 = 'Paused'
  1845 = 'Position hold'
  2517 = 'Position:'
  905 = 'Position: %s'
  731 = 'Powered on'
  1825 = 'Previous'
  316 = 'Program'
  1005 = 'Read to file'
  690 = 'Recipe list:'
  2365 = 'Recipe name'
  1499 = 'Recipe name:'
  247 = 'Recipe parameters'
  298 = 'Recipes'
  2656 = 'Recipes Manager: %s'
  1083 = 'Release'
  2097 = 'Reload'
  2954 = 'Remove'
  3075 = 'Reset'
  707 = 'Reset in progress...'
  861 = 'Reset:'
  1061 = 'Reseting errors...'
  561 = 'Restore'
  2648 = 'Restore auto'
  610 = 'Robot 1'
  951 = 'Robots'
  2584 = 'Safe Inputs'
  958 = 'Safe mode switch in progress...'
  711 = 'Safe mode switching...'
  1087 = 'Safe Outputs'
  670 = 'Safety I/O'
  2626 = 'Save in file'
  550 = 'Select'
  1288 = 'Selected recipe'
  7 = 'Selected recipe value'
  1458 = 'Selected recipe:'
  1007 = 'Service'
  2402 = 'Servo off'
  772 = 'Servo on'
  2183 = 'Set Position:'
  511 = 'Set Velocity:'
  536 = 'Severity'
  50 = 'Software version: v%s'
  450 = 'Start'
  3789 = 'Started'
  1037 = 'State: %s'
  895 = 'Status'
  85 = 'Statuses & parameters:'
  442 = 'Stop'
  1093 = 'Stopped'
  848 = 'Time Cleared'
  730 = 'Time Confirmed'
  9 = 'Time Raised'
  1974 = 'Time: %d [ms]'
  10 = 'Total active alarms'
  1629 = 'Update recipes'
  1334 = 'Velocity:'
  322 = '[%s/s]'
  374 = '[%s]'
END_TEXTLIST

// ---- VISUs/Alarms/EventTable.TcVIS
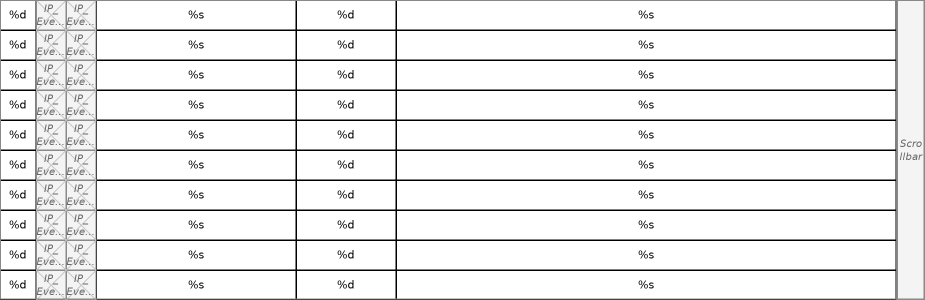
VISUALIZATION EventTable  // 925x300
VAR_IN_OUT
	data : ARRAY[1..512] OF ST_Event;
END_VAR
VAR 
	iIndex : INT;
END_VAR
    Group (0,0 896x30), invisible if: data[iIndex+1].iType = 0
        OnMouseClick: OpenDialog Dialog=SingleEvent, Parameters={data: data[iIndex+1]}, OpenModal=True, OpenCentered=True
        Rectangle (0,0 36x30), "%d", text variable: iIndex + 1
        Image (36,0 30x30), invisible if: data[iIndex+1].iType <> 1, image: IP_EventType.alarm
        Image (36,0 30x30), invisible if: data[iIndex+1].iType <> 2, image: IP_EventType.message
        Rectangle (96,0 200x30), "%s", text variable: LDT_TO_STRING(data[iIndex+1].iTimeStamp)
        Rectangle (296,0 100x30), "%d", text variable: data[iIndex+1].iEventId
        Image (66,0 30x30), invisible if: data[iIndex+1].eSeverity <> 4, image: IP_EventSeverity.critical
        Image (66,0 30x30), invisible if: data[iIndex+1].eSeverity <> 3, image: IP_EventSeverity.error
        Image (66,0 30x30), invisible if: data[iIndex+1].eSeverity <> 2, image: IP_EventSeverity.warning
        Image (66,0 30x30), invisible if: data[iIndex+1].eSeverity <> 1, image: IP_EventSeverity.info
        Image (66,0 30x30), invisible if: data[iIndex+1].eSeverity <> 0, image: IP_EventSeverity.verbose
        Rectangle (396,0 500x30), "%s", text variable: data[iIndex+1].sEventText
    Group (0,30 896x30), invisible if: data[iIndex+2].iType = 0
        OnMouseClick: OpenDialog Dialog=SingleEvent, Parameters={data: data[iIndex+2]}, OpenModal=True, OpenCentered=True
        Rectangle (0,0 36x30), "%d", text variable: iIndex + 2
        Image (36,0 30x30), invisible if: data[iIndex+2].iType <> 1, image: IP_EventType.alarm
        Image (36,0 30x30), invisible if: data[iIndex+2].iType <> 2, image: IP_EventType.message
        Rectangle (96,0 200x30), "%s", text variable: LDT_TO_STRING(data[iIndex+2].iTimeStamp)
        Rectangle (296,0 100x30), "%d", text variable: data[iIndex+2].iEventId
        Image (66,0 30x30), invisible if: data[iIndex+2].eSeverity <> 4, image: IP_EventSeverity.critical
        Image (66,0 30x30), invisible if: data[iIndex+2].eSeverity <> 3, image: IP_EventSeverity.error
        Image (66,0 30x30), invisible if: data[iIndex+2].eSeverity <> 2, image: IP_EventSeverity.warning
        Image (66,0 30x30), invisible if: data[iIndex+2].eSeverity <> 1, image: IP_EventSeverity.info
        Image (66,0 30x30), invisible if: data[iIndex+2].eSeverity <> 0, image: IP_EventSeverity.verbose
        Rectangle (396,0 500x30), "%s", text variable: data[iIndex+2].sEventText
    Group (0,60 896x30), invisible if: data[iIndex+3].iType = 0
        OnMouseClick: OpenDialog Dialog=SingleEvent, Parameters={data: data[iIndex+3]}, OpenModal=True, OpenCentered=True
        Rectangle (0,0 36x30), "%d", text variable: iIndex + 3
        Image (36,0 30x30), invisible if: data[iIndex+3].iType <> 1, image: IP_EventType.alarm
        Image (36,0 30x30), invisible if: data[iIndex+3].iType <> 2, image: IP_EventType.message
        Rectangle (96,0 200x30), "%s", text variable: LDT_TO_STRING(data[iIndex+3].iTimeStamp)
        Rectangle (296,0 100x30), "%d", text variable: data[iIndex+3].iEventId
        Image (66,0 30x30), invisible if: data[iIndex+3].eSeverity <> 4, image: IP_EventSeverity.critical
        Image (66,0 30x30), invisible if: data[iIndex+3].eSeverity <> 3, image: IP_EventSeverity.error
        Image (66,0 30x30), invisible if: data[iIndex+3].eSeverity <> 2, image: IP_EventSeverity.warning
        Image (66,0 30x30), invisible if: data[iIndex+3].eSeverity <> 1, image: IP_EventSeverity.info
        Image (66,0 30x30), invisible if: data[iIndex+3].eSeverity <> 0, image: IP_EventSeverity.verbose
        Rectangle (396,0 500x30), "%s", text variable: data[iIndex+3].sEventText
    Group (0,90 896x30), invisible if: data[iIndex+4].iType = 0
        OnMouseClick: OpenDialog Dialog=SingleEvent, Parameters={data: data[iIndex+4]}, OpenModal=True, OpenCentered=True
        Rectangle (0,0 36x30), "%d", text variable: iIndex + 4
        Image (36,0 30x30), invisible if: data[iIndex+4].iType <> 1, image: IP_EventType.alarm
        Image (36,0 30x30), invisible if: data[iIndex+4].iType <> 2, image: IP_EventType.message
        Rectangle (96,0 200x30), "%s", text variable: LDT_TO_STRING(data[iIndex+4].iTimeStamp)
        Rectangle (296,0 100x30), "%d", text variable: data[iIndex+4].iEventId
        Image (66,0 30x30), invisible if: data[iIndex+4].eSeverity <> 4, image: IP_EventSeverity.critical
        Image (66,0 30x30), invisible if: data[iIndex+4].eSeverity <> 3, image: IP_EventSeverity.error
        Image (66,0 30x30), invisible if: data[iIndex+4].eSeverity <> 2, image: IP_EventSeverity.warning
        Image (66,0 30x30), invisible if: data[iIndex+4].eSeverity <> 1, image: IP_EventSeverity.info
        Image (66,0 30x30), invisible if: data[iIndex+4].eSeverity <> 0, image: IP_EventSeverity.verbose
        Rectangle (396,0 500x30), "%s", text variable: data[iIndex+4].sEventText
    Group (0,120 896x30), invisible if: data[iIndex+5].iType = 0
        OnMouseClick: OpenDialog Dialog=SingleEvent, Parameters={data: data[iIndex+5]}, OpenModal=True, OpenCentered=True
        Rectangle (0,0 36x30), "%d", text variable: iIndex + 5
        Image (36,0 30x30), invisible if: data[iIndex+5].iType <> 1, image: IP_EventType.alarm
        Image (36,0 30x30), invisible if: data[iIndex+5].iType <> 2, image: IP_EventType.message
        Rectangle (96,0 200x30), "%s", text variable: LDT_TO_STRING(data[iIndex+5].iTimeStamp)
        Rectangle (296,0 100x30), "%d", text variable: data[iIndex+5].iEventId
        Image (66,0 30x30), invisible if: data[iIndex+5].eSeverity <> 4, image: IP_EventSeverity.critical
        Image (66,0 30x30), invisible if: data[iIndex+5].eSeverity <> 3, image: IP_EventSeverity.error
        Image (66,0 30x30), invisible if: data[iIndex+5].eSeverity <> 2, image: IP_EventSeverity.warning
        Image (66,0 30x30), invisible if: data[iIndex+5].eSeverity <> 1, image: IP_EventSeverity.info
        Image (66,0 30x30), invisible if: data[iIndex+5].eSeverity <> 0, image: IP_EventSeverity.verbose
        Rectangle (396,0 500x30), "%s", text variable: data[iIndex+5].sEventText
    Group (0,150 896x30), invisible if: data[iIndex+6].iType = 0
        OnMouseClick: OpenDialog Dialog=SingleEvent, Parameters={data: data[iIndex+6]}, OpenModal=True, OpenCentered=True
        Rectangle (0,0 36x30), "%d", text variable: iIndex + 6
        Image (36,0 30x30), invisible if: data[iIndex+6].iType <> 1, image: IP_EventType.alarm
        Image (36,0 30x30), invisible if: data[iIndex+6].iType <> 2, image: IP_EventType.message
        Rectangle (96,0 200x30), "%s", text variable: LDT_TO_STRING(data[iIndex+6].iTimeStamp)
        Rectangle (296,0 100x30), "%d", text variable: data[iIndex+6].iEventId
        Image (66,0 30x30), invisible if: data[iIndex+6].eSeverity <> 4, image: IP_EventSeverity.critical
        Image (66,0 30x30), invisible if: data[iIndex+6].eSeverity <> 3, image: IP_EventSeverity.error
        Image (66,0 30x30), invisible if: data[iIndex+6].eSeverity <> 2, image: IP_EventSeverity.warning
        Image (66,0 30x30), invisible if: data[iIndex+6].eSeverity <> 1, image: IP_EventSeverity.info
        Image (66,0 30x30), invisible if: data[iIndex+6].eSeverity <> 0, image: IP_EventSeverity.verbose
        Rectangle (396,0 500x30), "%s", text variable: data[iIndex+6].sEventText
    Group (0,180 896x30), invisible if: data[iIndex+7].iType = 0
        OnMouseClick: OpenDialog Dialog=SingleEvent, Parameters={data: data[iIndex+7]}, OpenModal=True, OpenCentered=True
        Rectangle (0,0 36x30), "%d", text variable: iIndex + 7
        Image (36,0 30x30), invisible if: data[iIndex+7].iType <> 1, image: IP_EventType.alarm
        Image (36,0 30x30), invisible if: data[iIndex+7].iType <> 2, image: IP_EventType.message
        Rectangle (96,0 200x30), "%s", text variable: LDT_TO_STRING(data[iIndex+7].iTimeStamp)
        Rectangle (296,0 100x30), "%d", text variable: data[iIndex+7].iEventId
        Image (66,0 30x30), invisible if: data[iIndex+7].eSeverity <> 4, image: IP_EventSeverity.critical
        Image (66,0 30x30), invisible if: data[iIndex+7].eSeverity <> 3, image: IP_EventSeverity.error
        Image (66,0 30x30), invisible if: data[iIndex+7].eSeverity <> 2, image: IP_EventSeverity.warning
        Image (66,0 30x30), invisible if: data[iIndex+7].eSeverity <> 1, image: IP_EventSeverity.info
        Image (66,0 30x30), invisible if: data[iIndex+7].eSeverity <> 0, image: IP_EventSeverity.verbose
        Rectangle (396,0 500x30), "%s", text variable: data[iIndex+7].sEventText
    Group (0,210 896x30), invisible if: data[iIndex+8].iType = 0
        OnMouseClick: OpenDialog Dialog=SingleEvent, Parameters={data: data[iIndex+8]}, OpenModal=True, OpenCentered=True
        Rectangle (0,0 36x30), "%d", text variable: iIndex + 8
        Image (36,0 30x30), invisible if: data[iIndex+8].iType <> 1, image: IP_EventType.alarm
        Image (36,0 30x30), invisible if: data[iIndex+8].iType <> 2, image: IP_EventType.message
        Rectangle (96,0 200x30), "%s", text variable: LDT_TO_STRING(data[iIndex+8].iTimeStamp)
        Rectangle (296,0 100x30), "%d", text variable: data[iIndex+8].iEventId
        Image (66,0 30x30), invisible if: data[iIndex+8].eSeverity <> 4, image: IP_EventSeverity.critical
        Image (66,0 30x30), invisible if: data[iIndex+8].eSeverity <> 3, image: IP_EventSeverity.error
        Image (66,0 30x30), invisible if: data[iIndex+8].eSeverity <> 2, image: IP_EventSeverity.warning
        Image (66,0 30x30), invisible if: data[iIndex+8].eSeverity <> 1, image: IP_EventSeverity.info
        Image (66,0 30x30), invisible if: data[iIndex+8].eSeverity <> 0, image: IP_EventSeverity.verbose
        Rectangle (396,0 500x30), "%s", text variable: data[iIndex+8].sEventText
    Group (0,240 896x30), invisible if: data[iIndex+9].iType = 0
        OnMouseClick: OpenDialog Dialog=SingleEvent, Parameters={data: data[iIndex+9]}, OpenModal=True, OpenCentered=True
        Rectangle (0,0 36x30), "%d", text variable: iIndex + 9
        Image (36,0 30x30), invisible if: data[iIndex+9].iType <> 1, image: IP_EventType.alarm
        Image (36,0 30x30), invisible if: data[iIndex+9].iType <> 2, image: IP_EventType.message
        Rectangle (96,0 200x30), "%s", text variable: LDT_TO_STRING(data[iIndex+9].iTimeStamp)
        Rectangle (296,0 100x30), "%d", text variable: data[iIndex+9].iEventId
        Image (66,0 30x30), invisible if: data[iIndex+9].eSeverity <> 4, image: IP_EventSeverity.critical
        Image (66,0 30x30), invisible if: data[iIndex+9].eSeverity <> 3, image: IP_EventSeverity.error
        Image (66,0 30x30), invisible if: data[iIndex+9].eSeverity <> 2, image: IP_EventSeverity.warning
        Image (66,0 30x30), invisible if: data[iIndex+9].eSeverity <> 1, image: IP_EventSeverity.info
        Image (66,0 30x30), invisible if: data[iIndex+9].eSeverity <> 0, image: IP_EventSeverity.verbose
        Rectangle (396,0 500x30), "%s", text variable: data[iIndex+9].sEventText
    Group (0,270 896x30), invisible if: data[iIndex+10].iType = 0
        OnMouseClick: OpenDialog Dialog=SingleEvent, Parameters={data: data[iIndex+10]}, OpenModal=True, OpenCentered=True
        Rectangle (0,0 36x30), "%d", text variable: iIndex + 10
        Image (36,0 30x30), invisible if: data[iIndex+10].iType <> 1, image: IP_EventType.alarm
        Image (36,0 30x30), invisible if: data[iIndex+10].iType <> 2, image: IP_EventType.message
        Rectangle (96,0 200x30), "%s", text variable: LDT_TO_STRING(data[iIndex+10].iTimeStamp)
        Rectangle (296,0 100x30), "%d", text variable: data[iIndex+10].iEventId
        Image (66,0 30x30), invisible if: data[iIndex+10].eSeverity <> 4, image: IP_EventSeverity.critical
        Image (66,0 30x30), invisible if: data[iIndex+10].eSeverity <> 3, image: IP_EventSeverity.error
        Image (66,0 30x30), invisible if: data[iIndex+10].eSeverity <> 2, image: IP_EventSeverity.warning
        Image (66,0 30x30), invisible if: data[iIndex+10].eSeverity <> 1, image: IP_EventSeverity.info
        Image (66,0 30x30), invisible if: data[iIndex+10].eSeverity <> 0, image: IP_EventSeverity.verbose
        Rectangle (396,0 500x30), "%s", text variable: data[iIndex+10].sEventText
    Scrollbar (897,0 28x300)
        p2245068023: GVL.iMAX_EVENTS - 10
        p1057716461: iIndex
END_VISUALIZATION

// ---- VISUs/Headers/Header.TcVIS
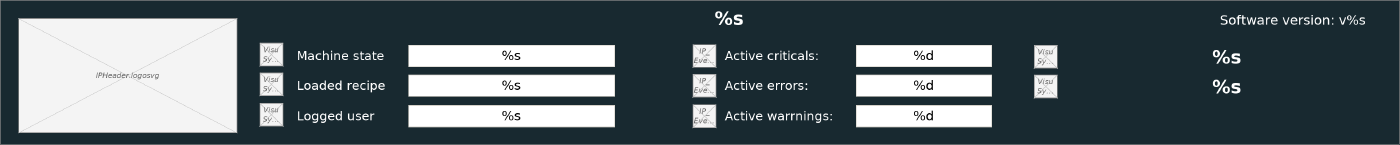
VISUALIZATION Header  // 1920x200
VAR_IN_OUT
	sMachineName		: STRING;					(*  *)
	sSoftwareVersion	: STRING;					(*  *)
	eMachineState		: E_MachineCtrlState;		(*  *)
	sCurrentRecipe		: STRING;					(*  *)
	sCurrentUser		: STRING;					(*  *)
	iActiveCriticals 	: UDINT;					(*  *)
	iActvieErrors		: UDINT;					(*  *)
	iActiveWarrnings	: UDINT;					(*  *)
	sCurrentDate		: STRING;					(*  *)
	sCurrentTime		: STRING;					(*  *)
END_VAR
    Label (404,59 133x36), "Machine state"
    Textfield (560,62 283x30), "%s", text list: 'TL_HeaderMachineState', text index: eMachineState
    Label (404,100 133x36), "Loaded recipe"
    Textfield (560,103 283x30), "%s", text variable: sCurrentRecipe
    Label (404,142 133x36), "Logged user"
    Textfield (560,145 283x30), "%s", text variable: sCurrentUser, text list: ''
    Label (991,59 133x36), "Active criticals:"
    Label (991,100 133x36), "Active errors:"
    Label (991,142 171x36), "Active warrnings:"
    Textfield (1174,62 186x30), "%d", text variable: iActiveCriticals
    Textfield (1174,103 186x30), "%d", text variable: iActvieErrors
    Textfield (1174,145 186x30), "%d", text variable: iActiveWarrnings
    Image (950,61 32x32), image: IP_EventSeverity.critical
    Image (950,102 32x32), image: IP_EventSeverity.error
    Image (950,144 32x32), image: IP_EventSeverity.warning
    Image (1418,62 32x32), image: VisuSymbols.Symbols.Calender
    Image (1418,103 32x32), image: VisuSymbols.Symbols.Clock
    Image (356,142 32x32), image: VisuSymbols.Symbols.User
    Image (356,59 32x32), image: VisuSymbols.Symbols.voltage
    Image (356,100 32x32), image: VisuSymbols.Symbols.Doc
    Textfield (700,10 600x30), "%s", text variable: sMachineName
    Textfield (1670,10 250x36), "Software version: v%s", text variable: sSoftwareVersion
    Textfield (1467,62 431x33), "%s", text variable: sCurrentDate
    Textfield (1467,103 431x33), "%s", text variable: sCurrentTime
    Image (25,25 300x158), image: IPHeader.logosvg
END_VISUALIZATION

// ---- VISUs/Headers/HeaderWinCE.TcVIS
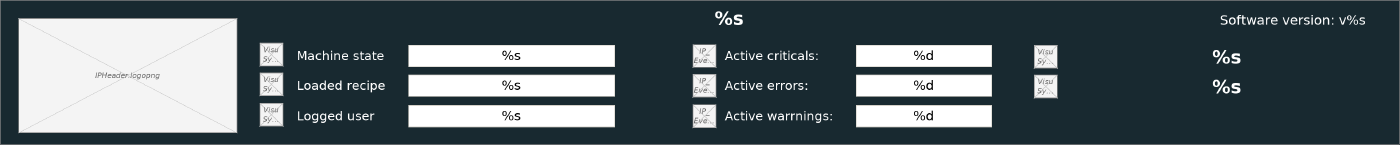
VISUALIZATION HeaderWinCE  // 1920x200
VAR_IN_OUT
	sMachineName		: STRING;					(*  *)
	sSoftwareVersion	: STRING;					(*  *)
	eMachineState		: E_MachineCtrlState;		(*  *)
	sCurrentRecipe		: STRING;					(*  *)
	sCurrentUser		: STRING;					(*  *)
	iActiveCriticals 	: UDINT;					(*  *)
	iActvieErrors		: UDINT;					(*  *)
	iActiveWarrnings	: UDINT;					(*  *)
	sCurrentDate		: STRING;					(*  *)
	sCurrentTime		: STRING;					(*  *)
END_VAR
    Label (404,59 133x36), "Machine state"
    Textfield (560,62 283x30), "%s", text list: 'TL_HeaderMachineState', text index: eMachineState
    Label (404,100 133x36), "Loaded recipe"
    Textfield (560,103 283x30), "%s", text variable: sCurrentRecipe
    Label (404,142 133x36), "Logged user"
    Textfield (560,145 283x30), "%s", text variable: sCurrentUser, text list: ''
    Label (991,59 133x36), "Active criticals:"
    Label (991,100 133x36), "Active errors:"
    Label (991,142 171x36), "Active warrnings:"
    Textfield (1174,62 186x30), "%d", text variable: iActiveCriticals
    Textfield (1174,103 186x30), "%d", text variable: iActvieErrors
    Textfield (1174,145 186x30), "%d", text variable: iActiveWarrnings
    Image (950,61 32x32), image: IP_EventSeverity.critical
    Image (950,102 32x32), image: IP_EventSeverity.error
    Image (950,144 32x32), image: IP_EventSeverity.warning
    Image (1418,62 32x32), image: VisuSymbols.Symbols.Calender
    Image (1418,103 32x32), image: VisuSymbols.Symbols.Clock
    Image (356,142 32x32), image: VisuSymbols.Symbols.User
    Image (356,59 32x32), image: VisuSymbols.Symbols.voltage
    Image (356,100 32x32), image: VisuSymbols.Symbols.Doc
    Textfield (700,10 600x30), "%s", text variable: sMachineName
    Textfield (1670,10 250x36), "Software version: v%s", text variable: sSoftwareVersion
    Textfield (1467,62 431x33), "%s", text variable: sCurrentDate
    Textfield (1467,103 431x33), "%s", text variable: sCurrentTime
    Image (25,25 300x158), image: IPHeader.logopng
END_VISUALIZATION

// ---- VISUs/Headers/Text Lists/TL_HeaderMachineState.TcTLO
TEXTLIST TL_HeaderMachineState
  0 = 'Uninitialized'
  10 = 'Initializing'
  20 = 'Ready-Initialized'
  30 = 'Auto'
  40 = 'Auto to Manual'
  50 = 'Manual'
  60 = 'Manual to Auto'
  70 = 'Reset'
  80 = 'Reset done'
  -10 = 'Aborting'
  -20 = 'Emergency'
   = ''
END_TEXTLIST

// ---- VISUs/Main.TcVIS
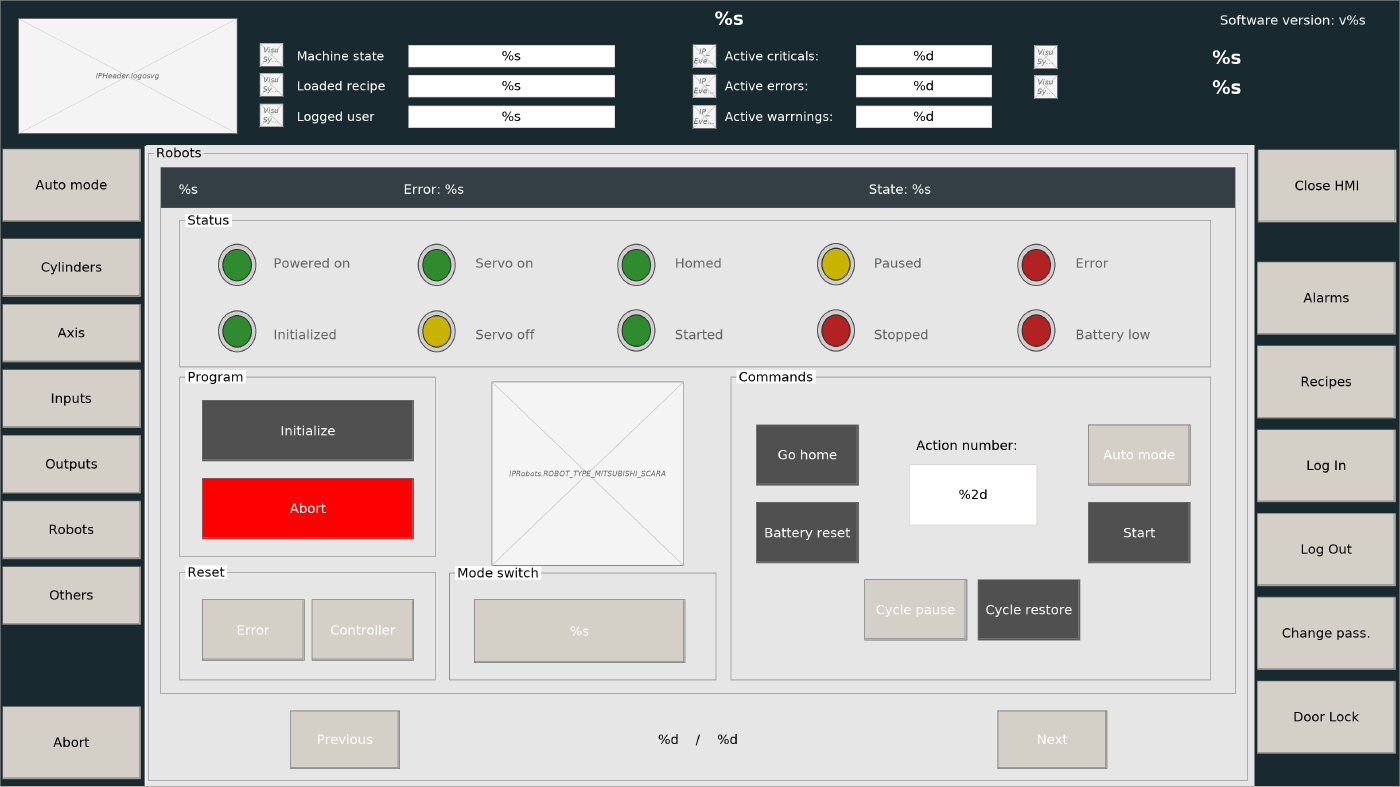
VISUALIZATION Main  // 1920x1080
    Frame (0,0 1920x200)
        shows Header(sMachineName := PRG_VisuControl.fbVisuControl.sMachineName, sSoftwareVersion := PRG_VisuControl.fbVisuControl.sSoftwareVersion, eMachineState := PRG_MachineControl.fbMachineControler.eMachineState, sCurrentRecipe := PRG_VisuControl.fbVisuControl.sCurrentRecipe, sCurrentUser := PRG_VisuControl.fbVisuControl.sCurrentUser, iActiveCriticals := PRG_VisuControl.fbVisuControl.iActiveCriticals, iActvieErrors := PRG_VisuControl.fbVisuControl.iActvieErrors, iActiveWarrnings := PRG_VisuControl.fbVisuControl.iActiveWarrnings, sCurrentDate := PRG_VisuControl.fbVisuControl.sCurrentDate, sCurrentTime := PRG_VisuControl.fbVisuControl.sCurrentTime)
    Frame (1720,199 200x880)
        shows NavBarAuxilary(btnAlarms := PRG_VisuControl.fbVisuControl.btnAlarms, btnRecipes := PRG_VisuControl.fbVisuControl.btnRecipes, btnDoorLock := PRG_VisuControl.fbVisuControl.btnLights, btnLogIn := PRG_VisuControl.fbVisuControl.btnLogIn, btnLogOut := PRG_VisuControl.fbVisuControl.btnLogOut, btnHmiClose := PRG_VisuControl.fbVisuControl.btnHmiClose, sCloseHMIFileName := PRG_VisuControl.fbVisuControl.sCloseHMIFileName, sCloseHMIParameters := PRG_VisuControl.fbVisuControl.sCloseHMIParameters, bVisNotInit := PRG_VisuControl.fbVisuControl.bVisNotInit, bVisHmiCLose := PRG_VisuControl.fbVisuControl.bVisHmiClose, bVisLogIn := PRG_VisuControl.fbVisuControl.bVisLogIn, bVisLogOut := PRG_VisuControl.fbVisuControl.bVisLogOut, bDoorLockDisabled := PRG_VisuControl.fbVisuControl.btnLights, bDoorLockInvisible := PRG_VisuControl.fbVisuControl.btnLights)
    Frame (200,199 1520x880)
        shows PageManualRobots(btnPrevious := PRG_VisuControl.fbVisuControl.btnPrevious, btnNext := PRG_VisuControl.fbVisuControl.btnNext, bPreviousInvisible := PRG_VisuControl.fbVisuControl.bPreviousInvisible, bNextInvisible := PRG_VisuControl.fbVisuControl.bNextInvisible, stRobotEmpty := PRG_VisuControl.fbVisuControl.arrRobotFrameEmpty[PRG_VisuControl.fbVisuControl.iSelectedRobotPageIndex], stRobot := PRG_VisuControl.fbVisuControl.arrRobotFrame[PRG_VisuControl.fbVisuControl.iSelectedRobotPageIndex], iRobotSelectedPageIndex := PRG_VisuControl.fbVisuControl.iSelectedRobotPageIndex, iRobotTotalPageIndex := PRG_VisuControl.fbVisuControl.iRobotPageIndex)
    Frame (-2,199 200x880)
        shows NavBarManual(btnAutoMode := PRG_VisuControl.fbVisuControl.btnAuto, btnCylinders := PRG_VisuControl.fbVisuControl.btnManualCylinder, btnMotors := PRG_VisuControl.fbVisuControl.btnManualAxis, btnSafety := PRG_VisuControl.fbVisuControl.btnManualSafety, btnInputs := PRG_VisuControl.fbVisuControl.btnManualInputs, btnOutputs := PRG_VisuControl.fbVisuControl.btnManualOutputs, btnOthers := PRG_VisuControl.fbVisuControl.btnManualOthers, btnAbort := PRG_VisuControl.fbVisuControl.btnAbort, btnRobots := PRG_VisuControl.fbVisuControl.btnManualRobots)
END_VISUALIZATION

// ---- VISUs/Manual/SingleAxis.TcVIS
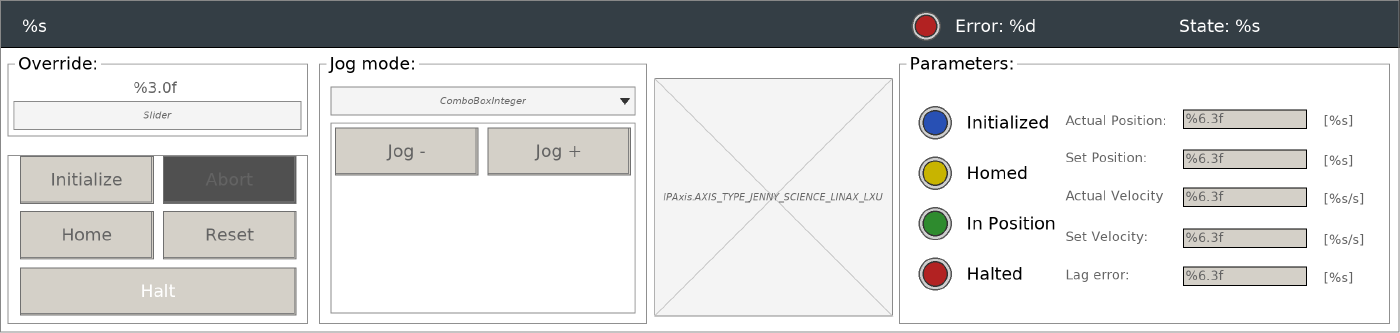
VISUALIZATION SingleAxis  // 1470x350
VAR_IN_OUT
	stAxis : ST_VisuCtrlAxisFrame;
END_VAR
    Rectangle (0,0 1470x50)
    Textfield (20,10 699x35), "%s", text variable: stAxis.sName
    Textfield (1235,10 225x35), "State: %s", text list: 'TL_SingleAxisState', text index: stAxis.eAxisState
    Lamp1 (955,10 35x35), variable: stAxis.bError, style: Lamp-Lamp1-Red
    Textfield (1000,10 200x35), "Error: %d", text variable: stAxis.iErrorID
    Image (687,82 250x250), image: IPAxis.AXIS_TYPE_JENNY_SCIENCE_LINAX_LXU
        p84334746: stAxis.sAxisImage
    GroupBox (8,59 315x84), "Override:"
        Slider (6,47 302x30), variable: stAxis.lrOverride, scale 0..100
        Rectangle (55,18 200x30), "%3.0f", text variable: stAxis.lrOverride
    GroupBox (8,155 315x185)
        Button (13,9 140x50), "Initialize"
            tap stAxis.btnInit
        Button (163,9 140x50), "Abort"
            tap stAxis.btnAbort
        Button (13,67 140x50), "Home"
            tap stAxis.btnHome
        Button (163,67 140x50), "Reset"
            tap stAxis.btnReset
        Button (13,126 290x50), "Halt"
            tap stAxis.btnHalt
    GroupBox (335,59 344x281), "Jog mode:"
        Frame (12,70 320x200), frame switch variable: stAxis.eJogMode
            shows SingleAxisJogStandardSlow(btnJogPositive := stAxis.btnJogPositive, btnJogNegative := stAxis.btnJogNegative)
            shows SingleAxisJogStandardFlast(btnJogPositive := stAxis.btnJogPositive, btnJogNegative := stAxis.btnJogNegative)
            shows SingleAxisJogContinous(btnJogPositive := stAxis.btnJogPositive, btnJogNegative := stAxis.btnJogNegative, lrVelocity := stAxis.lrJogVelocity, lrAcceleration := stAxis.lrJogAcceleration, lrDeceleration := stAxis.lrJogDeceleartion, sUnit := stAxis.sUnit)
            shows SingleAxisJogInching(btnJogPositive := stAxis.btnJogPositive, btnJogNegative := stAxis.btnJogNegative, lrPosition := stAxis.lrJogDistance, lrVelocity := stAxis.lrJogVelocity, lrAcceleration := stAxis.lrJogAcceleration, lrDeceleration := stAxis.lrJogDeceleartion, sUnit := stAxis.sUnit)
            shows SingleAxisJogInchingModulo(btnJogPositive := stAxis.btnJogPositive, btnJogNegative := stAxis.btnJogNegative, lrPosition := stAxis.lrJogDistance, lrVelocity := stAxis.lrJogVelocity, lrAcceleration := stAxis.lrJogAcceleration, lrDeceleration := stAxis.lrJogDeceleartion, sUnit := stAxis.sUnit)
        ComboBoxInteger (12,32 320x30), variable: stAxis.eJogMode, text list: 'TL_SingleAxisJogMode'
            p1601986498: ''
    GroupBox (944,59 515x281), "Parameters:"
        Rectangle (298,56 130x20), "%6.3f", text variable: stAxis.lrActualPosition
        Rectangle (443,59 62x18), "[%s]", text variable: stAxis.sUnit
        Rectangle (172,58 110x20), "Actual Position:"
        Lamp1 (18,156 40x40), variable: stAxis.bInPosition, style: Lamp-Lamp1-Green
        Lamp1 (18,50 40x40), variable: stAxis.bActive, style: Lamp-Lamp1-Blue
        Lamp1 (18,103 40x40), variable: stAxis.bHomed, style: Lamp-Lamp1-Yellow
        Label (68,55 100x30), "Initialized"
        Label (68,108 100x30), "Homed"
        Label (68,161 100x30), "In Position"
        Label (68,214 100x30), "Halted"
        Lamp1 (18,209 40x40), variable: stAxis.bHalted, style: Lamp-Lamp1-Red
        Rectangle (172,97 110x20), "Set Position:"
        Rectangle (298,98 130x20), "%6.3f", text variable: stAxis.lrSetPosition
        Rectangle (443,101 62x18), "[%s]", text variable: stAxis.sUnit
        Rectangle (172,137 110x20), "Actual Velocity"
        Rectangle (298,138 130x20), "%6.3f", text variable: stAxis.lrActualVelocity
        Rectangle (443,141 62x18), "[%s/s]", text variable: stAxis.sUnit
        Rectangle (172,180 110x20), "Set Velocity:"
        Rectangle (298,181 130x20), "%6.3f", text variable: stAxis.lrSetVelocity
        Rectangle (443,184 62x18), "[%s/s]", text variable: stAxis.sUnit
        Rectangle (172,220 110x20), "Lag error:"
        Rectangle (298,221 130x20), "%6.3f", text variable: stAxis.lrLagError
        Rectangle (443,224 62x18), "[%s]", text variable: stAxis.sUnit
END_VISUALIZATION

// ---- VISUs/Manual/SingleFixture.TcVIS
VISUALIZATION SingleFixture  // 1120x220
END_VISUALIZATION

// ---- VISUs/Manual/SingleAxisJogInching.TcVIS
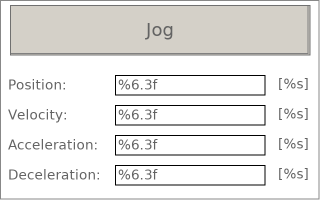
VISUALIZATION SingleAxisJogInching  // 320x200
VAR_IN_OUT
	btnJogPositive	: BOOL;
	btnJogNegative	: BOOL;
	lrPosition		: LREAL;
	lrVelocity		: LREAL;
	lrAcceleration	: LREAL;
	lrDeceleration	: LREAL;
	sUnit			: STRING;
END_VAR
    Rectangle (5,75 110x20), "Position:"
    Rectangle (115,75 150x20), "%6.3f", text variable: lrPosition
        OnMouseClick: write the text variable via VisuDialogs.Numpad
    Rectangle (275,75 44x18), "[%s]", text variable: sUnit
    Button (10,5 300x50), "Jog"
        tap btnJogPositive
    Rectangle (5,105 110x20), "Velocity:"
    Rectangle (115,105 150x20), "%6.3f", text variable: lrVelocity
        OnMouseClick: write the text variable via VisuDialogs.Numpad
    Rectangle (275,105 44x18), "[%s]", text variable: sUnit
    Rectangle (5,135 110x20), "Acceleration:"
    Rectangle (115,135 150x20), "%6.3f", text variable: lrAcceleration
        OnMouseClick: write the text variable via VisuDialogs.Numpad
    Rectangle (275,135 44x18), "[%s]", text variable: sUnit
    Rectangle (5,165 110x20), "Deceleration:"
    Rectangle (115,165 150x20), "%6.3f", text variable: lrDeceleration
        OnMouseClick: write the text variable via VisuDialogs.Numpad
    Rectangle (275,165 44x18), "[%s]", text variable: sUnit
END_VISUALIZATION

// ---- VISUs/Manual/SingleAxisJogContinous.TcVIS
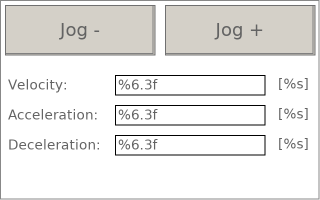
VISUALIZATION SingleAxisJogContinous  // 320x200
VAR_IN_OUT
	btnJogPositive	: BOOL;
	btnJogNegative	: BOOL;
	lrVelocity		: LREAL;
	lrAcceleration	: LREAL;
	lrDeceleration	: LREAL;
	sUnit			: STRING;
END_VAR
    Rectangle (5,75 110x20), "Velocity:"
    Rectangle (115,75 150x20), "%6.3f", text variable: lrVelocity
        OnMouseClick: write the text variable via VisuDialogs.Numpad
    Rectangle (275,75 44x18), "[%s]", text variable: sUnit
    Button (5,5 150x50), "Jog -"
        tap btnJogNegative
        OnMouseUp: toggle btnJogNegative
        OnMouseDown: toggle btnJogNegative
    Button (165,5 150x50), "Jog +"
        tap btnJogPositive
    Rectangle (5,105 110x20), "Acceleration:"
    Rectangle (115,105 150x20), "%6.3f", text variable: lrAcceleration
        OnMouseClick: write the text variable via VisuDialogs.Numpad
    Rectangle (275,105 44x18), "[%s]", text variable: sUnit
    Rectangle (5,135 110x20), "Deceleration:"
    Rectangle (115,135 150x20), "%6.3f", text variable: lrDeceleration
        OnMouseClick: write the text variable via VisuDialogs.Numpad
    Rectangle (275,135 44x18), "[%s]", text variable: sUnit
END_VISUALIZATION

// ---- VISUs/Manual/SingleAxisJogInchingModulo.TcVIS
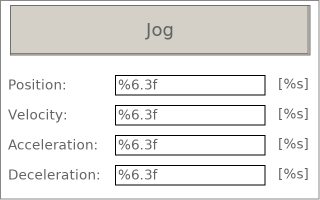
VISUALIZATION SingleAxisJogInchingModulo  // 320x200
VAR_IN_OUT
	btnJogPositive	: BOOL;
	btnJogNegative	: BOOL;
	lrPosition		: LREAL;
	lrVelocity		: LREAL;
	lrAcceleration	: LREAL;
	lrDeceleration	: LREAL;
	sUnit			: STRING;
END_VAR
    Rectangle (5,75 110x20), "Position:"
    Rectangle (115,75 150x20), "%6.3f", text variable: lrPosition
        OnMouseClick: write the text variable via VisuDialogs.Numpad
    Rectangle (275,75 44x18), "[%s]", text variable: sUnit
    Button (10,5 300x50), "Jog"
        tap btnJogPositive
    Rectangle (5,105 110x20), "Velocity:"
    Rectangle (115,105 150x20), "%6.3f", text variable: lrVelocity
        OnMouseClick: write the text variable via VisuDialogs.Numpad
    Rectangle (275,105 44x18), "[%s]", text variable: sUnit
    Rectangle (5,135 110x20), "Acceleration:"
    Rectangle (115,135 150x20), "%6.3f", text variable: lrAcceleration
        OnMouseClick: write the text variable via VisuDialogs.Numpad
    Rectangle (275,135 44x18), "[%s]", text variable: sUnit
    Rectangle (5,165 110x20), "Deceleration:"
    Rectangle (115,165 150x20), "%6.3f", text variable: lrDeceleration
        OnMouseClick: write the text variable via VisuDialogs.Numpad
    Rectangle (275,165 44x18), "[%s]", text variable: sUnit
END_VISUALIZATION

// ---- VISUs/Manual/SingleAxisJogStandardSlow.TcVIS
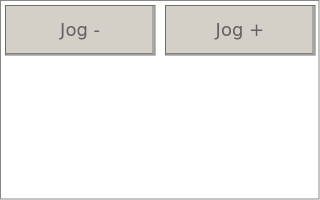
VISUALIZATION SingleAxisJogStandardSlow  // 320x200
VAR_IN_OUT
	btnJogPositive	: BOOL;
	btnJogNegative	: BOOL;
END_VAR
    Button (5,5 150x50), "Jog -"
        tap btnJogNegative
    Button (165,5 150x50), "Jog +"
        tap btnJogPositive
END_VISUALIZATION

// ---- VISUs/Manual/SingleAxisJogStandardFlast.TcVIS
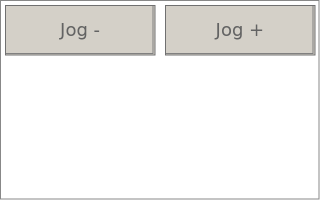
VISUALIZATION SingleAxisJogStandardFlast  // 320x200
VAR_IN_OUT
	btnJogPositive	: BOOL;
	btnJogNegative	: BOOL;
END_VAR
    Button (5,5 150x50), "Jog -"
        tap btnJogNegative
    Button (165,5 150x50), "Jog +"
        tap btnJogPositive
END_VISUALIZATION

// ---- VISUs/Manual/SingleCylinder.TcVIS
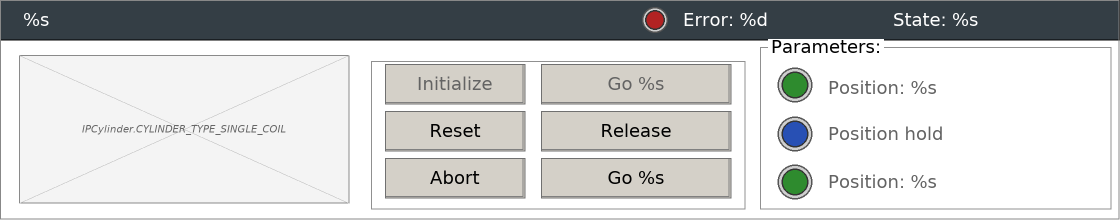
VISUALIZATION SingleCylinder  // 1120x220
VAR_IN_OUT
	stCylinder : ST_VisuCtrlCylinderFrame;
END_VAR
    Rectangle (0,0 1120x40)
    Textfield (20,5 524x30), "%s", text variable: stCylinder.sName
    Textfield (890,5 225x30), "State: %s", text list: 'TL_SingleCylinderState', text index: stCylinder.eCylinderState
    Lamp1 (640,5 30x30), variable: stCylinder.bError, style: Lamp-Lamp1-Red
    Textfield (680,5 200x30), "Error: %d", text variable: stCylinder.iErrorID
    GroupBox (760,39 351x170), "Parameters:"
        Rectangle (65,85 270x20), "Position hold", text variable: stCylinder.sHomeDescription
        Lamp1 (15,75 40x40), variable: stCylinder.bPositionHold, style: Lamp-Lamp1-Blue
        Rectangle (65,133 270x20), "Position: %s", text variable: stCylinder.sHomeDescription
        Rectangle (65,39 270x20), "Position: %s", text variable: stCylinder.sActiveDescription
        Lamp1 (15,26 40x40), variable: stCylinder.bSensorActive, style: Lamp-Lamp1-Green
        Lamp1 (15,123 40x40), variable: stCylinder.bSensorHome, style: Lamp-Lamp1-Green
    GroupBox (371,53 374x156)
        Button (170,105 190x40), "Go %s", text variable: stCylinder.sHomeDescription
            tap stCylinder.btnGoHome
        Button (170,58 190x40), "Release"
            tap stCylinder.btnRealase
        Button (170,11 190x40), "Go %s", text variable: stCylinder.sActiveDescription
            tap stCylinder.btnGoActive
        Button (14,105 140x40), "Abort", text variable: stCylinder.sHomeDescription
            tap stCylinder.btnAbort
        Button (14,58 140x40), "Reset"
            tap stCylinder.btnReset
        Button (14,11 140x40), "Initialize", text variable: stCylinder.sActiveDescription
            tap stCylinder.btnInit
    Image (19,55 330x148), image: IPCylinder.CYLINDER_TYPE_SINGLE_COIL
        p84334746: stCylinder.sCylinderImage
END_VISUALIZATION

// ---- VISUs/Manual/SingleDigitalInput.TcVIS
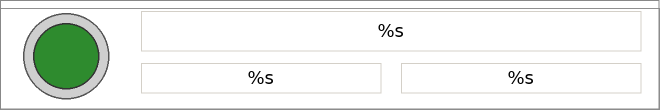
VISUALIZATION SingleDigitalInput  // 660x110
VAR_IN_OUT
	stDigitalInput : ST_VisuCtrlInputFrame;
END_VAR
    GroupBox (0,0 660x110)
        Lamp1 (16,6 100x100), variable: stDigitalInput.bIn, style: Lamp-Lamp1-Green
        Textfield (141,11 500x40), "%s", text variable: stDigitalInput.sName
        Textfield (141,63 240x30), "%s", text variable: stDigitalInput.sModuleType
        Textfield (401,63 240x30), "%s", text variable: stDigitalInput.sPortID
END_VISUALIZATION

// ---- VISUs/Manual/SingleRobot.TcVIS
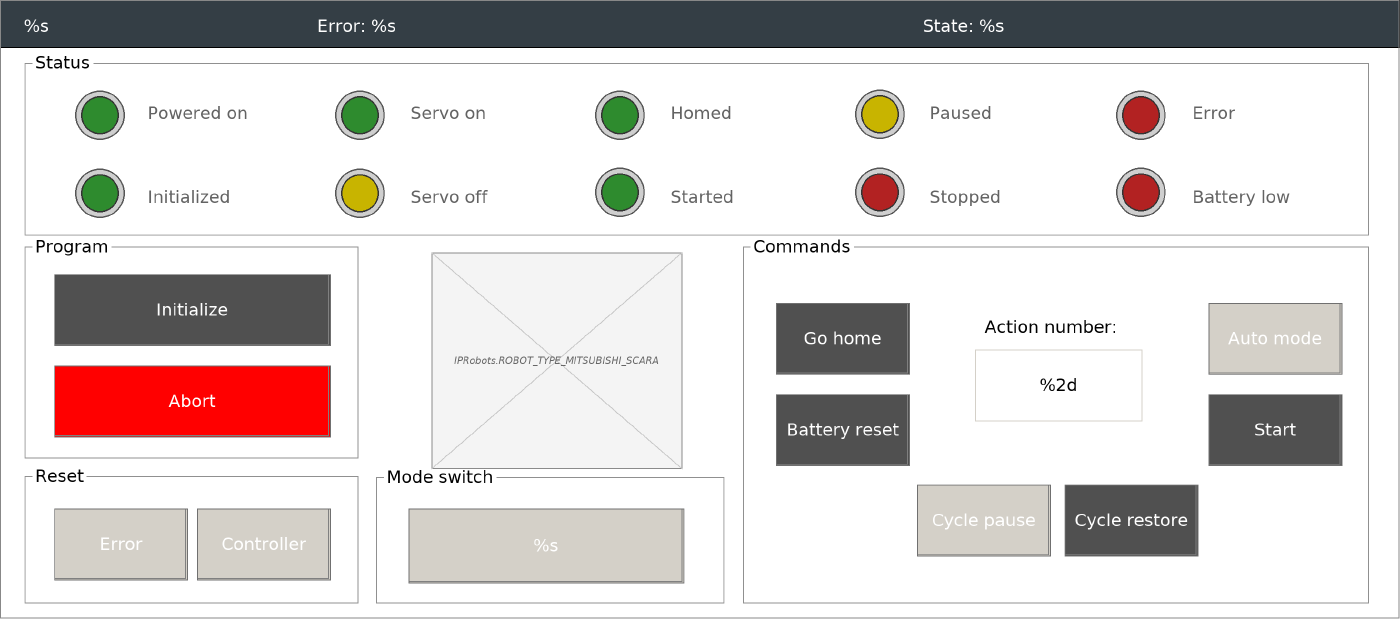
VISUALIZATION SingleRobot  // 1470x650
VAR_IN_OUT
	stRobot		: ST_VisuCtrlRobotFrame;
END_VAR
    Rectangle (0,0 1470x50)
    Textfield (22,10 296x35), "%s", text variable: stRobot.sName
    Textfield (966,10 498x35), "State: %s", text list: 'TL_SingleRobotState', text index: stRobot.eRobotState
    Textfield (330,10 628x35), "Error: %s", text variable: stRobot.sErrorDescription
    Image (453,265 263x227), image: IPRobots.ROBOT_TYPE_MITSUBISHI_SCARA
        p84334746: stRobot.sRobotImage
    GroupBox (26,58 1411x189), "Status"
        Lamp1 (595,33 60x60), variable: stRobot.bIsHomed, style: Lamp-Lamp1-Green
        Lamp1 (595,114 60x60), variable: stRobot.bStarted, style: Lamp-Lamp1-Green
        Rectangle (675,37 150x48), "Homed"
        Rectangle (675,125 150x48), "Started"
        Lamp1 (1142,114 60x60), variable: stRobot.bBatteryLow, style: Lamp-Lamp1-Red
        Rectangle (1223,125 150x48), "Battery low"
        Lamp1 (1142,33 60x60), variable: stRobot.bError, style: Lamp-Lamp1-Red
        Rectangle (1223,37 150x48), "Error"
        Lamp1 (49,33 60x60), variable: stRobot.bPowerOn, style: Lamp-Lamp1-Green
        Lamp1 (49,115 60x60), variable: stRobot.bInit, style: Lamp-Lamp1-Green
        Rectangle (126,37 150x48), "Powered on"
        Rectangle (126,125 150x48), "Initialized"
        Rectangle (402,37 150x48), "Servo on"
        Rectangle (402,125 150x48), "Servo off"
        Lamp1 (322,33 60x60), variable: stRobot.bServoOn, style: Lamp-Lamp1-Green
        Lamp1 (322,115 60x60), variable: stRobot.bServoOff, style: Lamp-Lamp1-Yellow
        Rectangle (947,37 150x48), "Paused"
        Rectangle (947,125 150x48), "Stopped"
        Lamp1 (868,32 60x60), variable: stRobot.bPaused, style: Lamp-Lamp1-Yellow
        Lamp1 (868,114 60x60), variable: stRobot.bStopped, style: Lamp-Lamp1-Red
    GroupBox (26,251 350x230), "Program"
        Button (31,37 290x75), "Initialize", input disabled if: stRobot.bInitButtonDisable
            tap stRobot.btnInit
        Button (31,133 290x75), "Abort", input disabled if: stRobot.bUninitialized
            tap stRobot.btnAbort
    GroupBox (26,492 350x141), "Reset"
        Button (31,42 140x75), "Error"
            tap stRobot.btnErrorReset
        Button (181,42 140x75), "Controller"
            tap stRobot.btnControllerReset
    GroupBox (780,251 657x382), "Commands"
        Button (489,163 140x75), "Start", input disabled if: stRobot.bActionButtonDisable
            tap stRobot.btnDoAction
        Button (35,67 140x75), "Go home", input disabled if: stRobot.bHomeButtonDisable
            tap stRobot.btnGoHome
        Button (489,67 140x75), "Auto mode", input disabled if: stRobot.bAutoButtonDisable
            tap stRobot.btnGoAuto
        Button (35,163 140x75), "Battery reset", input disabled if: stRobot.bAutoButtonDisable
        Rectangle (251,80 160x25), "Action number:"
        Button (338,258 140x75), "Cycle restore", input disabled if: stRobot.bRestoreCycleButtonDisable
            tap stRobot.btnRestoreCycle
        Button (183,258 140x75), "Cycle pause", input disabled if: stRobot.bPausingButtonDisable
            tap stRobot.btnCyclePause
        Textfield (244,116 175x75), "%2d", text variable: stRobot.iActionNumber, input disabled if: stRobot.bActionButtonDisable
            OnMouseClick: write the text variable via VisuDialogs.Numpad, min 13, max 100
    GroupBox (395,493 365x140), "Mode switch", invisible if: stRobot.bModeSwitchButtonDisabled
        Button (34,41 289x78), "%s", input disabled if: stRobot.bInit, text list: 'TL_ModeSwitchState', text index: stRobot.bModeSwitchState
            toggle stRobot.btnModeSwitch
END_VISUALIZATION

// ---- VISUs/Manual/SingleSafeOutput.TcVIS
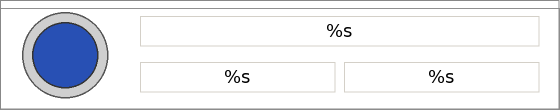
VISUALIZATION SingleSafeOutput  // 560x110
VAR_IN_OUT
	stDigitalOutput : ST_VisuCtrlOutputFrame;
END_VAR
    GroupBox (0,0 560x110)
        Lamp1 (15,5 100x100), variable: stDigitalOutput.bOut, style: Lamp-Lamp1-Blue
        Textfield (344,62 195x30), "%s", text variable: stDigitalOutput.sPortID
        Textfield (140,62 195x30), "%s", text variable: stDigitalOutput.sModuleType
        Textfield (140,16 399x30), "%s", text variable: stDigitalOutput.sName
END_VISUALIZATION

// ---- VISUs/Manual/SingleSafeInput.TcVIS
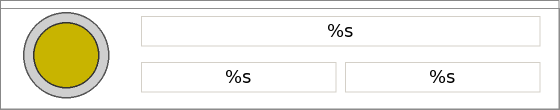
VISUALIZATION SingleSafeInput  // 560x110
VAR_IN_OUT
	stDigitalInput : ST_VisuCtrlInputFrame;
END_VAR
    GroupBox (0,0 560x110)
        Lamp1 (16,5 100x100), variable: stDigitalInput.bIn, style: Lamp-Lamp1-Yellow
        Textfield (141,16 399x30), "%s", text variable: stDigitalInput.sName
        Textfield (345,62 195x30), "%s", text variable: stDigitalInput.sPortID
        Textfield (141,62 195x30), "%s", text variable: stDigitalInput.sModuleType
END_VISUALIZATION

// ---- VISUs/Manual/SingleDigitalOutput.TcVIS
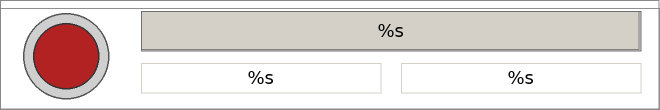
VISUALIZATION SingleDigitalOutput  // 660x110
VAR_IN_OUT
	stDigitalOutput : ST_VisuCtrlOutputFrame;
END_VAR
    GroupBox (0,0 660x110)
        Lamp1 (16,6 100x100), variable: stDigitalOutput.bOut, style: Lamp-Lamp1-Red
        Button (141,11 500x40), "%s", text variable: stDigitalOutput.sName, input disabled if: stDigitalOutput.bControlable, text list: ''
            toggle stDigitalOutput.btnOut
        Textfield (141,63 240x30), "%s", text variable: stDigitalOutput.sModuleType
        Textfield (401,63 240x30), "%s", text variable: stDigitalOutput.sPortID
END_VISUALIZATION

// ---- VISUs/Manual/Text Lists/TL_ModeSwitchState.TcTLO
TEXTLIST TL_ModeSwitchState
  0 = 'Auto'
  1 = 'Manual'
   = ''
END_TEXTLIST

// ---- VISUs/Manual/Text Lists/TL_SingleAxisJogMode.TcTLO
TEXTLIST TL_SingleAxisJogMode
  0 = 'Standard slow'
  1 = 'Standard fast'
  2 = 'Continous'
  3 = 'Inching'
  4 = 'Inching modulo'
   = ''
END_TEXTLIST

// ---- VISUs/Manual/Text Lists/TL_SingleCylinderState.TcTLO
TEXTLIST TL_SingleCylinderState
  0 = 'Uninitialized'
  10 = 'Initializing'
  20 = 'Ready initialized'
  30 = 'Idle'
  40 = 'Go active'
  50 = 'Go active done'
  60 = 'Go home'
  70 = 'Go home done'
  80 = 'Release'
  90 = 'Release done'
  100 = 'Reset'
  110 = 'Reset done'
  -10 = 'Aborting'
   = ''
END_TEXTLIST

// ---- VISUs/Manual/Text Lists/TL_SingleAxisState.TcTLO
TEXTLIST TL_SingleAxisState
  0 = 'Uninitialized\t'
  10 = 'Initializing'
  20 = 'Ready initialized'
  30 = 'Idle'
  40 = 'Home'
  50 = 'Home done'
  60 = 'Move velocity'
  70 = 'Move velocity done'
  80 = 'Move absolute'
  90 = 'Move absolute done'
  100 = 'Move additive'
  110 = 'Move additive done'
  120 = 'Move relative'
  130 = 'Move relative done'
  140 = 'Move jog'
  150 = 'Move jog done'
  160 = 'Stop'
  170 = 'Stop done'
  180 = 'Halt'
  190 = 'Halt done'
  200 = 'Reset'
  210 = 'Reset done'
  220 = 'Coupling'
  230 = 'Coupling done'
  240 = 'Decoupling'
  250 = 'Decoupling done'
  -10 = 'Aborting'
   = ''
END_TEXTLIST

// ---- VISUs/Manual/Text Lists/TL_SingleRobotState.TcTLO
TEXTLIST TL_SingleRobotState
  0 = 'Uninitialized\t'
  10 = 'Initializing'
  20 = 'Ready initialized'
  30 = 'Idle- not homed'
  40 = 'Going home'
  50 = 'Home done'
  60 = 'Idle homed'
  70 = 'Updating recipes'
  80 = 'Updating recipes done'
  100 = 'Going auto'
  110 = 'Going auto done'
  120 = 'Idle auto'
  130 = 'Doing action'
  140 = 'Doing action done'
  200 = 'Cycle stopping'
  210 = 'Cycle stopping done'
  220 = 'Idle auto paused'
  230 = 'Auto restoring'
  240 = 'Auto restoring done'
  300 = 'Cycle pausing'
  310 = 'Cycle pausing done'
  320 = 'Idle cycle paused'
  330 = 'Cycle restoring'
  340 = 'Cycle restoring done'
  500 = 'Reset'
  510 = 'Reset done'
  -10 = 'In external error'
  -20 = 'Aborting'
   = ''
END_TEXTLIST

// ---- VISUs/Navigation/NavBarAuto.TcVIS
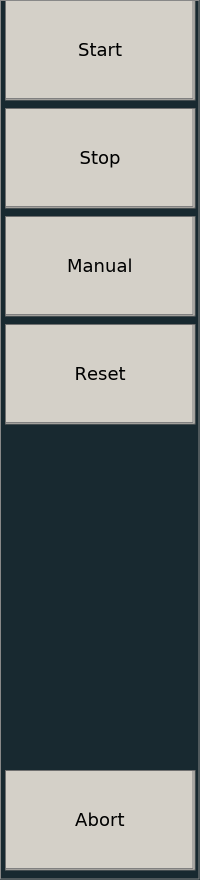
VISUALIZATION NavBarAuto  // 200x880
VAR_IN_OUT
	btnStart 		: BOOL;
	btnStop 		: BOOL;
	btnManualMode	: BOOL;
	btnAbort		: BOOL;
	btnReset		: BOOL;
	
	bVisStart 		: BOOL;
	bVisStop		: BOOL;
END_VAR
    Button (5,0 190x100), "Start", input disabled if: bVisStart
        tap btnStart
    Button (5,108 190x100), "Stop", input disabled if: bVisStop
        tap btnStop
    Button (5,770 190x100), "Abort", input disabled if: bVisStart
        tap btnAbort
    Button (5,216 190x100), "Manual", input disabled if: bVisStart
        tap btnManualMode
    Button (5,324 190x100), "Reset", input disabled if: bVisStart
        tap btnReset
END_VISUALIZATION

// ---- VISUs/Navigation/NavBarAuxilary.TcVIS
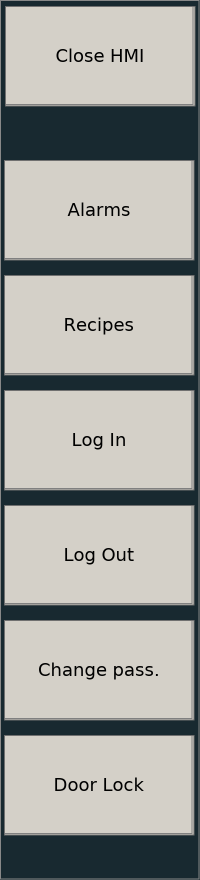
VISUALIZATION NavBarAuxilary  // 200x880
VAR_IN_OUT
	btnAlarms			: BOOL;
	btnRecipes			: BOOL;
	btnDoorLock			: BOOL;
	btnLogIn			: BOOL;
	btnLogOut			: BOOL;
	btnHmiClose			: BOOL;
	sCloseHMIFileName	: STRING;
	sCloseHMIParameters	: STRING;
	
	bVisNotInit 		: BOOL;
	bVisHmiCLose		: BOOL;
	bVisLogIn			: BOOL;
	bVisLogOut			: BOOL;
	bDoorLockDisabled	: BOOL;
	bDoorLockInvisible	: BOOL;
END_VAR
    Button (5,6 190x100), "Close HMI", input disabled if: bVisHmiCLose
        tap btnHmiClose
        toggle btnHmiClose
        OnMouseClick: ExecuteCommand ExecuteCommand=ExecuteCommand=[Command=ExecutePlcProgram, Value=sCloseHMIFileName, Value2=sCloseHMIParameters, Command=ExecutePlcProgram]
    Button (4,390 190x100), "Log In", input disabled if: bVisLogIn
        tap btnLogIn
        OnMouseUp: VisuUserMgmt Type=Login
    Button (4,505 190x100), "Log Out", input disabled if: bVisLogOut
        tap btnLogOut
        OnMouseUp: VisuUserMgmt Type=Logout
    Button (4,620 190x100), "Change pass.", input disabled if: bVisLogOut
        OnMouseUp: VisuUserMgmt Type=ChangeUserPassword
    Button (4,160 190x100), "Alarms"
        tap btnAlarms
    Button (4,275 190x100), "Recipes", input disabled if: bVisNotInit
        tap btnRecipes
    Button (4,735 190x100), "Door Lock", invisible if: bDoorLockInvisible, input disabled if: bDoorLockDisabled
        toggle btnDoorLock
END_VISUALIZATION

// ---- VISUs/Navigation/NavBarEmpty.TcVIS
VISUALIZATION NavBarEmpty  // 200x880
END_VISUALIZATION

// ---- VISUs/Navigation/NavBarInitializing.TcVIS
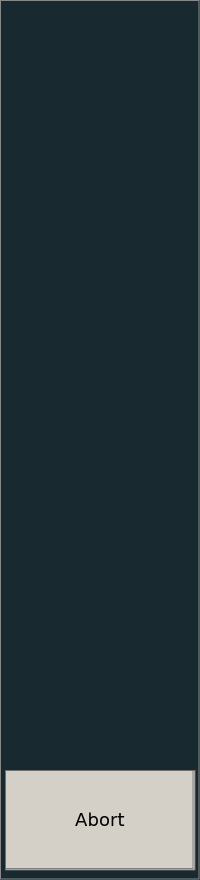
VISUALIZATION NavBarInitializing  // 200x880
VAR_IN_OUT
	btnAbort : BOOL;
END_VAR
    Button (5,770 190x100), "Abort"
        tap btnAbort
END_VISUALIZATION

// ---- VISUs/Navigation/NavBarManual.TcVIS
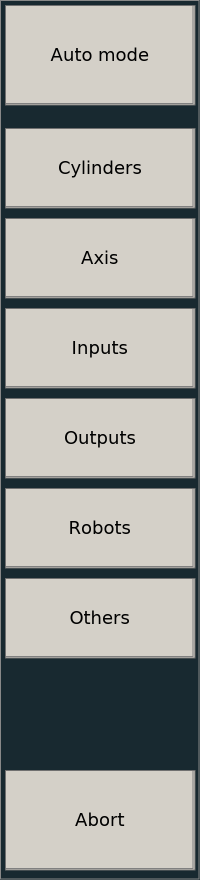
VISUALIZATION NavBarManual  // 200x880
VAR_IN_OUT
	btnAutoMode	: BOOL;
	btnCylinders: BOOL;
	btnMotors	: BOOL;
	btnSafety	: BOOL;
	btnInputs	: BOOL;
	btnOutputs	: BOOL;
	btnOthers	: BOOL;
	btnAbort	: BOOL;
	btnRobots 	: BOOL;
END_VAR
    Button (5,128 190x80), "Cylinders"
        tap btnCylinders
    Button (5,218 190x80), "Axis"
        tap btnMotors
    Button (5,770 190x100), "Abort"
        tap btnAbort
    Button (5,398 190x80), "Outputs"
        tap btnOutputs
    Button (5,308 190x80), "Inputs"
        tap btnInputs
    Button (5,5 190x100), "Auto mode"
        tap btnAutoMode
    Button (5,578 190x80), "Others"
        tap btnOthers
    Button (5,488 190x80), "Robots"
        tap btnRobots
END_VISUALIZATION

// ---- VISUs/Navigation/NavBarUninitialized.TcVIS
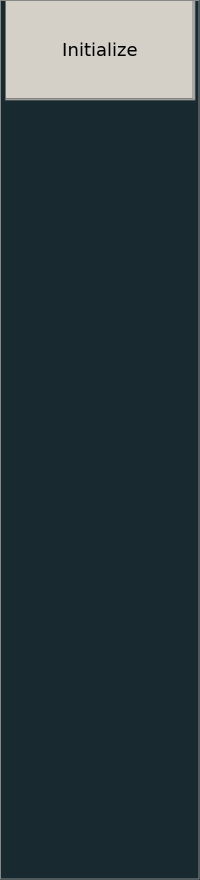
VISUALIZATION NavBarUninitialized  // 200x880
VAR_IN_OUT
	btnInitialize	: BOOL;	(*  *)
END_VAR
    Button (5,0 190x100), "Initialize"
        tap btnInitialize
END_VISUALIZATION

// ---- VISUs/Navigation/NavBarUtilities.TcVIS
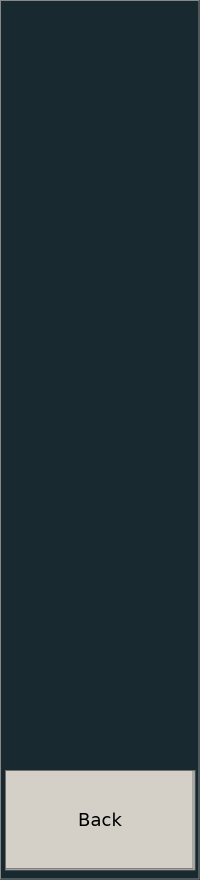
VISUALIZATION NavBarUtilities  // 200x880
VAR_IN_OUT
	btnBack : BOOL;
END_VAR
    Button (5,770 190x100), "Back"
        tap btnBack
END_VISUALIZATION

// ---- VISUs/Pages/PageInitializing.TcVIS
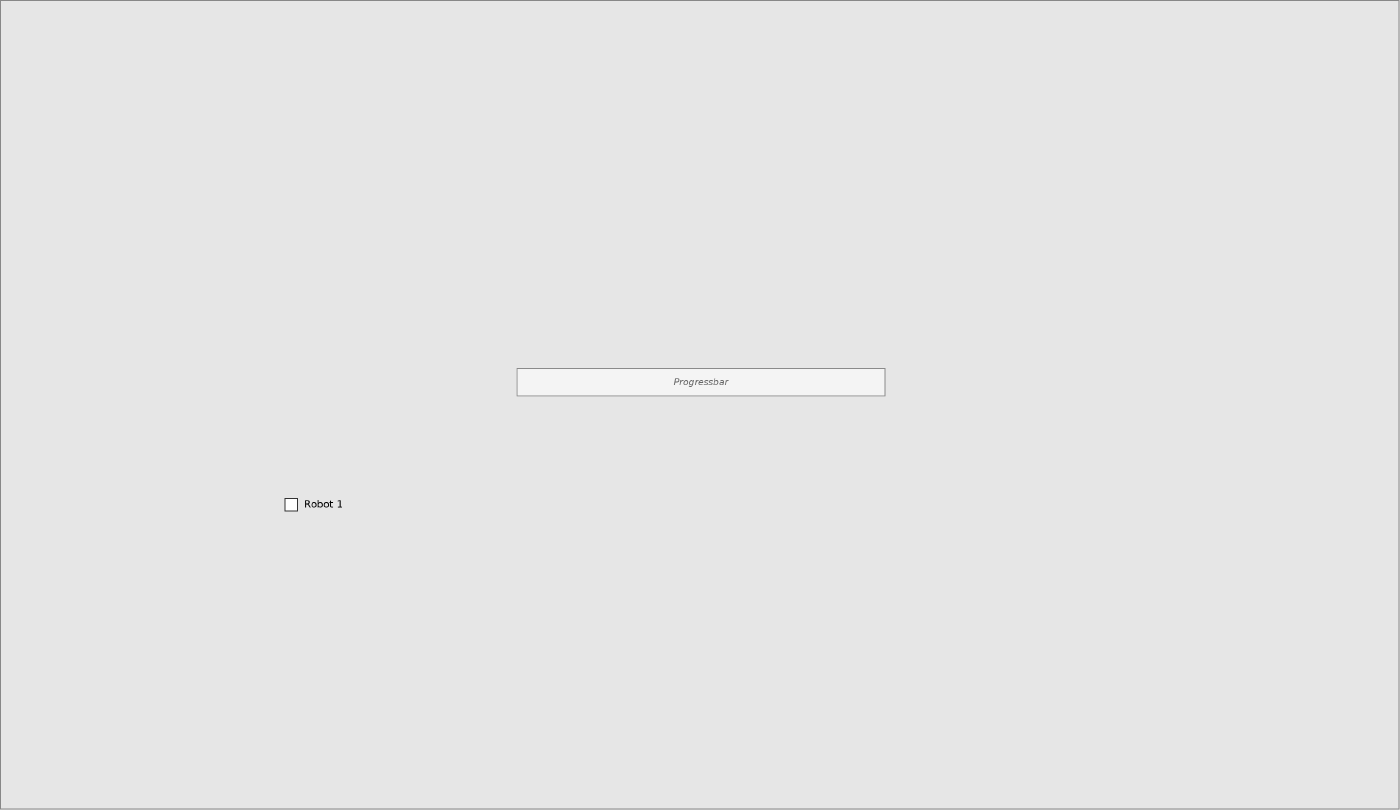
VISUALIZATION PageInitializing  // 1520x880
    Progressbar (561,400 400x30)
    Checkbox (307,533 320x30), "Robot 1"
END_VISUALIZATION

// ---- VISUs/Pages/PageXtsEnviroment.TcVIS
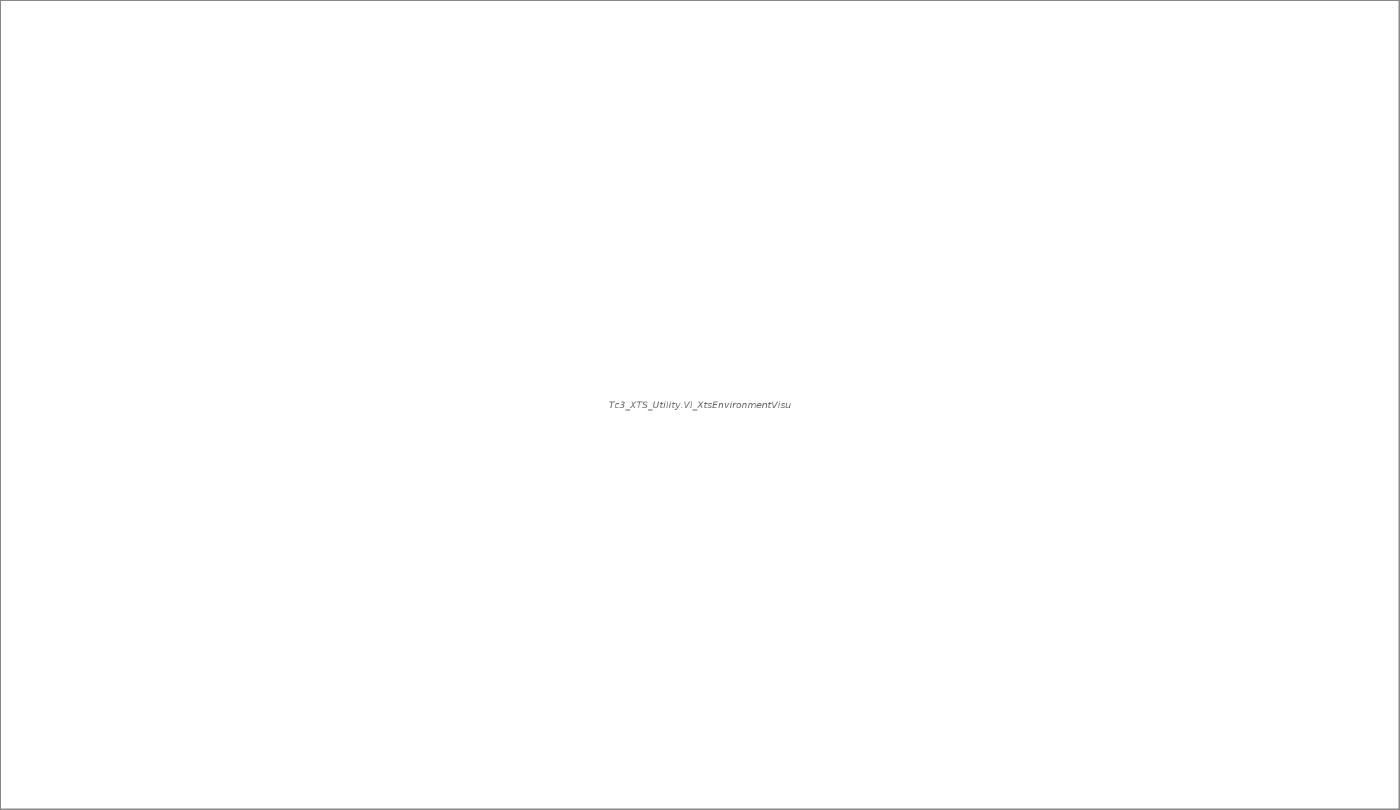
VISUALIZATION PageXtsEnviroment  // 1520x880
    Frame (0,0 1520x880)
        shows Tc3_XTS_Utility.VI_XtsEnvironmentVisu()
END_VISUALIZATION

// ---- VISUs/Pages/PageAborting.TcVIS
